// assign actuator mode
      AN    M    120.1;
      =     DB2740.DBX  105.4;
      =     DB2740.DBX  185.4;
      S     DB2740.DBX  265.4;
      =     DB2740.DBX  345.4;
      =     DB2740.DBX  425.4;
      =     DB2740.DBX  505.4;
      =     DB2740.DBX  585.4;
      =     DB2740.DBX  665.4;
      =     DB2740.DBX  745.4;
      =     DB2740.DBX  825.4;
      =     DB2740.DBX  905.4;
      =     DB2740.DBX  985.4;
      =     DB2740.DBX 1065.4;
      =     DB2740.DBX 1145.4;
      =     DB2740.DBX 1225.4;
      =     DB2740.DBX 1305.4;
      =     DB2740.DBX 1385.4;
      =     DB2740.DBX 1465.4;
      =     DB2740.DBX 1545.4;
      =     DB2740.DBX 1625.4;
      =     DB2740.DBX 1705.4;
      =     DB2740.DBX 1785.4;
      =     DB2740.DBX 1865.4;
      =     DB2740.DBX 1945.4;
      =     DB2740.DBX 2025.4;
      =     DB2740.DBX 2105.4;
      =     DB2740.DBX 2185.4;
      =     DB2740.DBX 2265.4;
      =     DB2740.DBX 2345.4;
      =     DB2740.DBX 2425.4;
      =     DB2740.DBX 2505.4;
      =     DB2740.DBX 2585.4;
      =     DB2740.DBX 2665.4;

MODE: SET   ;

NETWORK
TITLE =A14RRP1 Reinigungsrücklaufpumpe Anlage 14
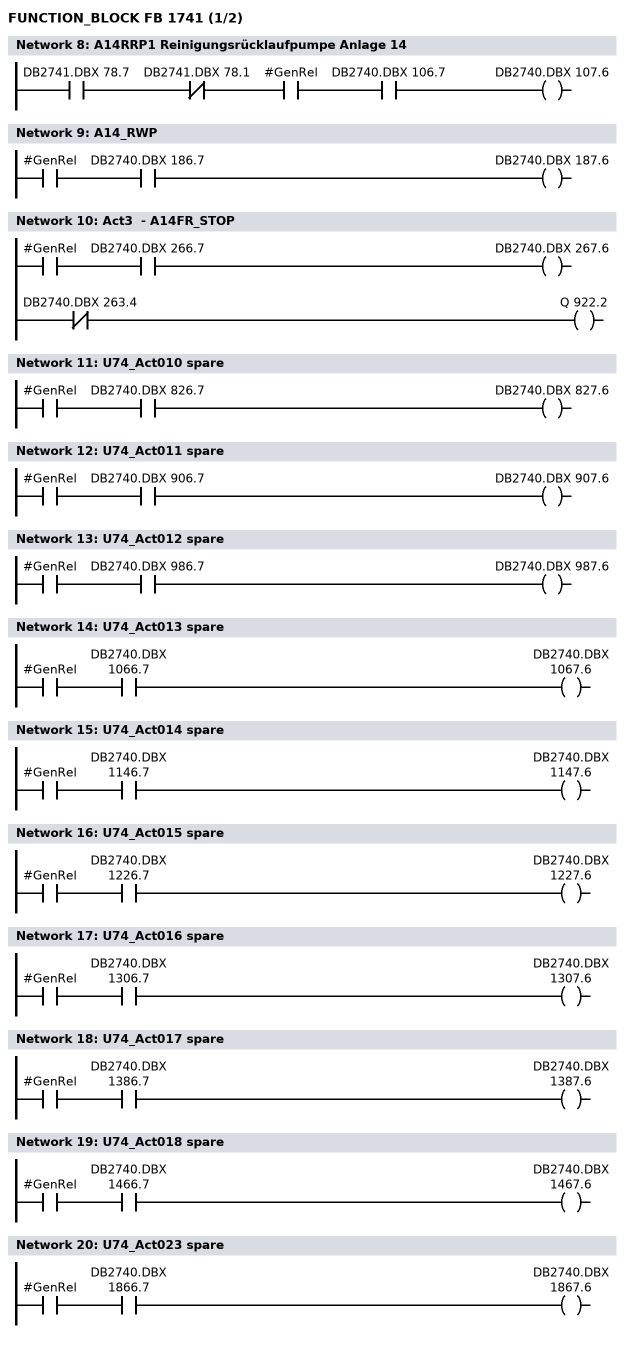

      A     DB2741.DBX   78.7;
      AN    DB2741.DBX   78.1;

      A     #GenRel;
      A     DB2740.DBX  106.7;
      =     DB2740.DBX  107.6;
NETWORK
TITLE =A14_RWP

      A     #GenRel;
      A     DB2740.DBX  186.7;
      =     DB2740.DBX  187.6;

NETWORK
TITLE =Act3  - A14FR_STOP

      A     #GenRel;
      A     DB2740.DBX  266.7;
      =     DB2740.DBX  267.6;

      AN    DB2740.DBX  263.4;
      =     Q    922.2;
NETWORK
TITLE =U74_Act010 spare

      A     #GenRel;
      A     DB2740.DBX  826.7;
      =     DB2740.DBX  827.6;
NETWORK
TITLE =U74_Act011 spare

      A     #GenRel;
      A     DB2740.DBX  906.7;
      =     DB2740.DBX  907.6;
NETWORK
TITLE =U74_Act012 spare

      A     #GenRel;
      A     DB2740.DBX  986.7;
      =     DB2740.DBX  987.6;
NETWORK
TITLE =U74_Act013 spare

      A     #GenRel;
      A     DB2740.DBX 1066.7;
      =     DB2740.DBX 1067.6;
NETWORK
TITLE =U74_Act014 spare

      A     #GenRel;
      A     DB2740.DBX 1146.7;
      =     DB2740.DBX 1147.6;
NETWORK
TITLE =U74_Act015 spare

      A     #GenRel;
      A     DB2740.DBX 1226.7;
      =     DB2740.DBX 1227.6;
NETWORK
TITLE =U74_Act016 spare

      A     #GenRel;
      A     DB2740.DBX 1306.7;
      =     DB2740.DBX 1307.6;
NETWORK
TITLE =U74_Act017 spare

      A     #GenRel;
      A     DB2740.DBX 1386.7;
      =     DB2740.DBX 1387.6;
NETWORK
TITLE =U74_Act018 spare

      A     #GenRel;
      A     DB2740.DBX 1466.7;
      =     DB2740.DBX 1467.6;
NETWORK
TITLE =U74_Act023 spare

      A     #GenRel;
      A     DB2740.DBX 1866.7;
      =     DB2740.DBX 1867.6;
NETWORK
TITLE =U74_Act024 spare
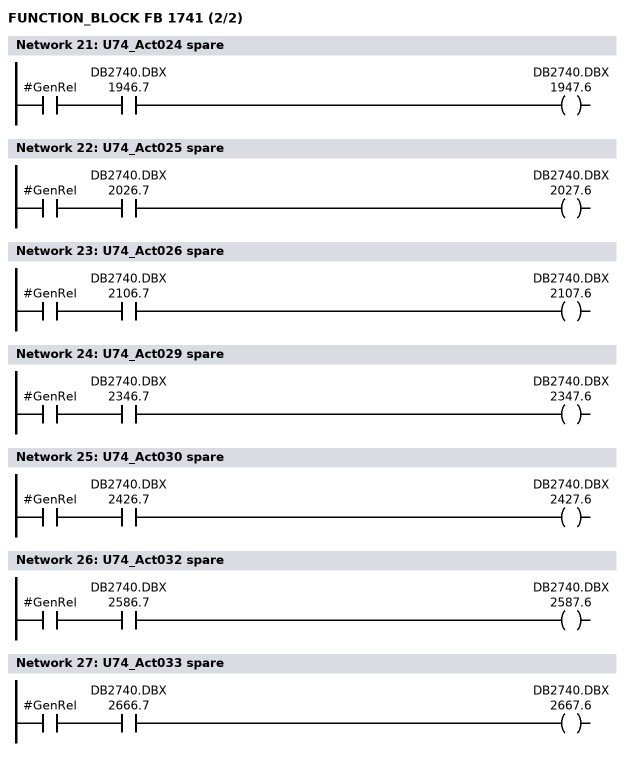

      A     #GenRel;
      A     DB2740.DBX 1946.7;
      =     DB2740.DBX 1947.6;
NETWORK
TITLE =U74_Act025 spare

      A     #GenRel;
      A     DB2740.DBX 2026.7;
      =     DB2740.DBX 2027.6;
NETWORK
TITLE =U74_Act026 spare

      A     #GenRel;
      A     DB2740.DBX 2106.7;
      =     DB2740.DBX 2107.6;
NETWORK
TITLE =U74_Act029 spare

      A     #GenRel;
      A     DB2740.DBX 2346.7;
      =     DB2740.DBX 2347.6;
NETWORK
TITLE =U74_Act030 spare

      A     #GenRel;
      A     DB2740.DBX 2426.7;
      =     DB2740.DBX 2427.6;
NETWORK
TITLE =U74_Act032 spare

      A     #GenRel;
      A     DB2740.DBX 2586.7;
      =     DB2740.DBX 2587.6;
NETWORK
TITLE =U74_Act033 spare

      A     #GenRel;
      A     DB2740.DBX 2666.7;
      =     DB2740.DBX 2667.6;
END_FUNCTION_BLOCK

FUNCTION_BLOCK FB 1770
TITLE =U077: KZE Anlage  3
FAMILY : BOTEC_F1
NAME : U077A
VERSION : 2.1


VAR_TEMP
  EStopOK : BOOL ;	//auxiliary flag
  CIP : BOOL ;	//CIP Program Selected
  xTmp : BOOL ;	//Temporary Bool(free for general use)
  DummyBool : BOOL ;	//Temporary Bool(free for general use)
  UnitNo : INT ;	//unit number
  UnitFB : INT ;	//unit expansion FB number
  rTmp : REAL ;	//Temporary REAL (free for general use)
  iTmp : INT ;	//Temporary INT (free for general use)
  DummyInt : INT ;	//Temporary INT (free for general use)
  dTmp : DINT ;	//Temporary DINT (free for general use)
END_VAR
BEGIN
NETWORK
TITLE =general

      CLR   ;
      =     #xTmp;
      =     #EStopOK;

      L     DB1770.DBW    0;
      T     #UnitNo;
      L     DB1770.DBW    2;
      T     #UnitFB;

NETWORK
TITLE =Universal value

      NOP   0;
// unv001 UnV 001 Process Status
      CALL FC    27 (
           UnitNo                   := #UnitNo,
           UnVRec                   := DB2775.unv001,
           ValExt                   := DB2775.DBD  234);

// unv002 UnV 002 Universal Value 02
      CALL FC    27 (
           UnitNo                   := #UnitNo,
           UnVRec                   := DB2775.unv002,
           ValExt                   := DB2775.DBD  362);

// unv003 UnV 003 Universal Value 03
      CALL FC    27 (
           UnitNo                   := #UnitNo,
           UnVRec                   := DB2775.unv003,
           ValExt                   := DB2775.DBD  490);

// unv004 UnV 004 Universal Value 04
      CALL FC    27 (
           UnitNo                   := #UnitNo,
           UnVRec                   := DB2775.unv004,
           ValExt                   := DB2775.DBD  618);

NETWORK
TITLE =special inputs

      NOP   0;
// KEG_MIXER_BOGEN_23_24 SpI 001 KEG Mixer/KZE Schwenkbogen
      CALL FC    14 (
           UnitNo                   := #UnitNo,
           SpIRec                   := DB2771.KEG_MIXER_BOGEN_23_24,
           SpIBit                   := I    950.0);

// KEG_MIXER_BOGEN_25_26 SpI 002 KEG Mixer/KZE Schwenkbogen
      CALL FC    14 (
           UnitNo                   := #UnitNo,
           SpIRec                   := DB2771.KEG_MIXER_BOGEN_25_26,
           SpIBit                   := I    950.1);

// KEG_MIXER_BOGEN_27_28 SpI 003 KEG Mixer/KZE Schwenkbogen
      CALL FC    14 (
           UnitNo                   := #UnitNo,
           SpIRec                   := DB2771.KEG_MIXER_BOGEN_27_28,
           SpIBit                   := I    950.2);

// KEG_MIXER_BOGEN_27_28_30 SpI 004 KEG Mixer/KZE Schwenkbogen
      CALL FC    14 (
           UnitNo                   := #UnitNo,
           SpIRec                   := DB2771.KEG_MIXER_BOGEN_27_28_30,
           SpIBit                   := I    950.3);

// KEG_MIXER_BOGEN_29_32 SpI 005 KEG Mixer/KZE Schwenkbogen
      CALL FC    14 (
           UnitNo                   := #UnitNo,
           SpIRec                   := DB2771.KEG_MIXER_BOGEN_29_32,
           SpIBit                   := I    950.4);

// KEG_MIXER_BOGEN_31_32 SpI 006 KEG Mixer/KZE Schwenkbogen
      CALL FC    14 (
           UnitNo                   := #UnitNo,
           SpIRec                   := DB2771.KEG_MIXER_BOGEN_31_32,
           SpIBit                   := I    950.5);

// KEG_MIXER_BOGEN_31_33 SpI 007 KEG Mixer/KZE Schwenkbogen
      CALL FC    14 (
           UnitNo                   := #UnitNo,
           SpIRec                   := DB2771.KEG_MIXER_BOGEN_31_33,
           SpIBit                   := I    950.6);

// KEG_MIXER_BOGEN_34_38 SpI 008 KEG Mixer/KZE Schwenkbogen
      CALL FC    14 (
           UnitNo                   := #UnitNo,
           SpIRec                   := DB2771.KEG_MIXER_BOGEN_34_38,
           SpIBit                   := I    950.7);

// KEG_MIXER_BOGEN_35_36_40 SpI 009 KEG Mixer/KZE Schwenkbogen
      CALL FC    14 (
           UnitNo                   := #UnitNo,
           SpIRec                   := DB2771.KEG_MIXER_BOGEN_35_36_40,
           SpIBit                   := I    951.0);

// KEG_MIXER_BOGEN_37_41 SpI 010 KEG Mixer/KZE Schwenkbogen
      CALL FC    14 (
           UnitNo                   := #UnitNo,
           SpIRec                   := DB2771.KEG_MIXER_BOGEN_37_41,
           SpIBit                   := I    951.1);

// KEG_MIXER_BOGEN_21_22 SpI 011 KEG Mixer/KZE Schwenkbogen
      CALL FC    14 (
           UnitNo                   := #UnitNo,
           SpIRec                   := DB2771.KEG_MIXER_BOGEN_21_22,
           SpIBit                   := I    951.2);

// KEG_MIXER_BOGEN_22_24 SpI 012 KEG Mixer/KZE Schwenkbogen
      CALL FC    14 (
           UnitNo                   := #UnitNo,
           SpIRec                   := DB2771.KEG_MIXER_BOGEN_22_24,
           SpIBit                   := I    951.3);

// KEG_MIXER_BOGEN_27_30 SpI 013 KEG Mixer/KZE Schwenkbogen
      CALL FC    14 (
           UnitNo                   := #UnitNo,
           SpIRec                   := DB2771.KEG_MIXER_BOGEN_27_30,
           SpIBit                   := I    951.4);

// KEG_MIXER_FRG_KZE SpI 014 KEG Mixer/KZE Freigabe CIP nur KZE
      CALL FC    14 (
           UnitNo                   := #UnitNo,
           SpIRec                   := DB2771.KEG_MIXER_FRG_KZE,
           SpIBit                   := I    947.0);

// KEG_MIXER_FRG_GES SpI 015 KEG Mixer/KZE Freigabe CIP Gesamt
      CALL FC    14 (
           UnitNo                   := #UnitNo,
           SpIRec                   := DB2771.KEG_MIXER_FRG_GES,
           SpIBit                   := I    946.6);

// KEG_MIXER_FRG_o_KZE SpI 016 KEG Mixer/KZE Freigabe CIP Gesamt ohne KZE
      CALL FC    14 (
           UnitNo                   := #UnitNo,
           SpIRec                   := DB2771.KEG_MIXER_FRG_o_KZE,
           SpIBit                   := I    946.7);

// KEG_MIXER_BOGEN_28_31 SpI 020 KEG Mixer/KZE Schwenkbogen
      CALL FC    14 (
           UnitNo                   := #UnitNo,
           SpIRec                   := DB2771.KEG_MIXER_BOGEN_28_31,
           SpIBit                   := I    951.5);

NETWORK
TITLE =messages

      NOP   0;
// msg001 Msg 001 Message 01
      CALL FC    16 (
           UnitNo                   := #UnitNo,
           MsgRec                   := DB2777.msg001,
           MsgBit                   := DB2777.DBX   82.7);

// msg002 Msg 002 Message 02
      CALL FC    16 (
           UnitNo                   := #UnitNo,
           MsgRec                   := DB2777.msg002,
           MsgBit                   := DB2777.DBX  142.7);

// msg003 Msg 003 Message 03
      CALL FC    16 (
           UnitNo                   := #UnitNo,
           MsgRec                   := DB2777.msg003,
           MsgBit                   := DB2777.DBX  202.7);

NETWORK
TITLE =unit supply

      UC    FB [#UnitFB];
END_FUNCTION_BLOCK

FUNCTION_BLOCK FB 1771
TITLE =U077: KZE Anlage  3
FAMILY : BOTEC_F1
NAME : U077E
VERSION : 1.2


VAR_TEMP
  CIP : BOOL ;	//CIP active
  UNIM : BOOL ;	//Unit Not In Maintenance
  GenRel : BOOL ;	//general OK (emergency and maintenance OK)
  EStopOK : BOOL ;	//emergency OK
  UnitNo : INT ;	//unit number
  xTmp : BOOL ;	//Temporary Bool
  iTmp : INT ;	//Temporary INT
  rTmp : REAL ;	//Temporary REAL
  dTmp : DINT ;	//Temporary DINT (free for general use)
  RetValInt : INT ;	//return value
END_VAR
BEGIN
NETWORK
TITLE =General

      SET   ;
// Simulation ---------------------------------------------------------------
      A     DB1771.DBX 1357.7;
      CC    FB  1779; // "U077Sim"
      A     DB1771.DBX   17.3;
      =     DB1771.DBX 1357.7; //Help bit for simulation

// get unit number ----------------------------------------------------------
      L     DB1770.DBW    0;
      T     #UnitNo;

// CIP ----------------------------------------------------------------------
      L     DB1771.DBD   54;
      L     0;
      <D    ;
      =     #CIP;

// emergency OK -------------------------------------------------------------
      A     DB1775.DBX   27.0; //Emergency Stop OK
      =     #EStopOK;

// Write Unit in Maintenance ------------------------------------------------

      AN    DB1771.DBX   69.7;
      =     #UNIM;

// emergency and maintenance OK ---------------------------------------------
      A     #EStopOK;
      A     #UNIM;
      =     #GenRel;

// communication ------------------------------------------------------------
      UC    FB  1775; // U077Com

NETWORK
TITLE =Universal Value

      NOP   0;

// ----------------------------------------------------------
// unv001 Process Status
// ----------------------------------------------------------
// process value to UnV
//      L     0.000000e+000
//      T     "U077UnVD".unv001.ValExt

// ----------------------------------------------------------
// unv002 Universal Value 02
// ----------------------------------------------------------
// process value to UnV
//      L     0.000000e+000
//      T     "U077UnVD".unv002.ValExt

// ----------------------------------------------------------
// unv003 Universal Value 03
// ----------------------------------------------------------
// process value to UnV
//      L     0.000000e+000
//      T     "U077UnVD".unv003.ValExt

// ----------------------------------------------------------
// unv004 Universal Value 04
// ----------------------------------------------------------
// process value to UnV
//      L     0.000000e+000
//      T     "U077UnVD".unv004.ValExt

NETWORK
TITLE =Special Input

      NOP   0;

// ----------------------------------------------------------
// KEG_MIXER_BOGEN_23_24 KEG Mixer/KZE Schwenkbogen
// ----------------------------------------------------------
//      SET
//      =     "U077SpID".KEG_MIXER_BOGEN_23_24.EAl
//      =     "U077SpID".KEG_MIXER_BOGEN_23_24.Pre

// ----------------------------------------------------------
// KEG_MIXER_BOGEN_25_26 KEG Mixer/KZE Schwenkbogen
// ----------------------------------------------------------
//      SET
//      =     "U077SpID".KEG_MIXER_BOGEN_25_26.EAl
//      =     "U077SpID".KEG_MIXER_BOGEN_25_26.Pre

// ----------------------------------------------------------
// KEG_MIXER_BOGEN_27_28 KEG Mixer/KZE Schwenkbogen
// ----------------------------------------------------------
//      SET
//      =     "U077SpID".KEG_MIXER_BOGEN_27_28.EAl
//      =     "U077SpID".KEG_MIXER_BOGEN_27_28.Pre

// ----------------------------------------------------------
// KEG_MIXER_BOGEN_27_28_30 KEG Mixer/KZE Schwenkbogen
// ----------------------------------------------------------
//      SET
//      =     "U077SpID".KEG_MIXER_BOGEN_27_28_30.EAl
//      =     "U077SpID".KEG_MIXER_BOGEN_27_28_30.Pre

// ----------------------------------------------------------
// KEG_MIXER_BOGEN_29_32 KEG Mixer/KZE Schwenkbogen
// ----------------------------------------------------------
//      SET
//      =     "U077SpID".KEG_MIXER_BOGEN_29_32.EAl
//      =     "U077SpID".KEG_MIXER_BOGEN_29_32.Pre

// ----------------------------------------------------------
// KEG_MIXER_BOGEN_31_32 KEG Mixer/KZE Schwenkbogen
// ----------------------------------------------------------
//      SET
//      =     "U077SpID".KEG_MIXER_BOGEN_31_32.EAl
//      =     "U077SpID".KEG_MIXER_BOGEN_31_32.Pre

// ----------------------------------------------------------
// KEG_MIXER_BOGEN_31_33 KEG Mixer/KZE Schwenkbogen
// ----------------------------------------------------------
//      SET
//      =     "U077SpID".KEG_MIXER_BOGEN_31_33.EAl
//      =     "U077SpID".KEG_MIXER_BOGEN_31_33.Pre

// ----------------------------------------------------------
// KEG_MIXER_BOGEN_34_38 KEG Mixer/KZE Schwenkbogen
// ----------------------------------------------------------
//      SET
//      =     "U077SpID".KEG_MIXER_BOGEN_34_38.EAl
//      =     "U077SpID".KEG_MIXER_BOGEN_34_38.Pre

// ----------------------------------------------------------
// KEG_MIXER_BOGEN_35_36_40 KEG Mixer/KZE Schwenkbogen
// ----------------------------------------------------------
//      SET
//      =     "U077SpID".KEG_MIXER_BOGEN_35_36_40.EAl
//      =     "U077SpID".KEG_MIXER_BOGEN_35_36_40.Pre

// ----------------------------------------------------------
// KEG_MIXER_BOGEN_37_41 KEG Mixer/KZE Schwenkbogen
// ----------------------------------------------------------
//      SET
//      =     "U077SpID".KEG_MIXER_BOGEN_37_41.EAl
//      =     "U077SpID".KEG_MIXER_BOGEN_37_41.Pre

// ----------------------------------------------------------
// KEG_MIXER_BOGEN_21_22 KEG Mixer/KZE Schwenkbogen
// ----------------------------------------------------------
//      SET
//      =     "U077SpID".KEG_MIXER_BOGEN_21_22.EAl
//      =     "U077SpID".KEG_MIXER_BOGEN_21_22.Pre

// ----------------------------------------------------------
// KEG_MIXER_BOGEN_22_24 KEG Mixer/KZE Schwenkbogen
// ----------------------------------------------------------
//      SET
//      =     "U077SpID".KEG_MIXER_BOGEN_22_24.EAl
//      =     "U077SpID".KEG_MIXER_BOGEN_22_24.Pre

// ----------------------------------------------------------
// KEG_MIXER_BOGEN_27_30 KEG Mixer/KZE Schwenkbogen
// ----------------------------------------------------------
//      SET
//      =     "U077SpID".KEG_MIXER_BOGEN_27_30.EAl
//      =     "U077SpID".KEG_MIXER_BOGEN_27_30.Pre

// ----------------------------------------------------------
// KEG_MIXER_FRG_KZE KEG Mixer/KZE Freigabe CIP nur KZE
// ----------------------------------------------------------
//      SET
//      =     "U077SpID".KEG_MIXER_FRG_KZE.EAl
//      =     "U077SpID".KEG_MIXER_FRG_KZE.Pre

// ----------------------------------------------------------
// KEG_MIXER_FRG_GES KEG Mixer/KZE Freigabe CIP Gesamt
// ----------------------------------------------------------
//      SET
//      =     "U077SpID".KEG_MIXER_FRG_GES.EAl
//      =     "U077SpID".KEG_MIXER_FRG_GES.Pre

// ----------------------------------------------------------
// KEG_MIXER_FRG_o_KZE KEG Mixer/KZE Freigabe CIP Gesamt ohne KZE
// ----------------------------------------------------------
//      SET
//      =     "U077SpID".KEG_MIXER_FRG_o_KZE.EAl
//      =     "U077SpID".KEG_MIXER_FRG_o_KZE.Pre

// ----------------------------------------------------------
// KEG_MIXER_BOGEN_28_31 KEG Mixer/KZE Schwenkbogen
// ----------------------------------------------------------
//      SET
//      =     "U077SpID".KEG_MIXER_BOGEN_28_31.EAl
//      =     "U077SpID".KEG_MIXER_BOGEN_28_31.Pre

NETWORK
TITLE =Messages

      NOP   0;

// ----------------------------------------------------------
// msg001 Message 01
// ----------------------------------------------------------
      SET   ;
      R     DB2777.DBX   80.7;
      =     DB2777.DBX   81.4;

      CLR   ;
      =     DB2777.DBX   82.7;

// ----------------------------------------------------------
// msg002 Message 02
// ----------------------------------------------------------
      SET   ;
      R     DB2777.DBX  140.7;
      =     DB2777.DBX  141.4;

      CLR   ;
      =     DB2777.DBX  142.7;

// ----------------------------------------------------------
// msg003 Message 03
// ----------------------------------------------------------
      SET   ;
      R     DB2777.DBX  200.7;
      =     DB2777.DBX  201.4;

      CLR   ;
      =     DB2777.DBX  202.7;

NETWORK
TITLE =Sequence organisation

      CLR   ;
      =     M    122.2;

// SFM supply ----------------------------------------------------------------

// sequencer ----------------------------------------------------------------
      A     DB1773.DBX   43.1;
      S     DB1773.DBX   97.3;

      CALL FC    40 (
           UnitNo                   := #UnitNo);

NETWORK
TITLE =Auto / Manual

      SET   ;
      AN    M    122.2;
      JC    MODE;
      AN    M    120.1;




MODE: SET   ;

END_FUNCTION_BLOCK

FUNCTION_BLOCK FB 1780
TITLE =U078: KZE Anlage  5
FAMILY : BOTEC_F1
NAME : U078A
VERSION : 2.1


VAR_TEMP
  EStopOK : BOOL ;	//auxiliary flag
  CIP : BOOL ;	//CIP Program Selected
  xTmp : BOOL ;	//Temporary Bool(free for general use)
  DummyBool : BOOL ;	//Temporary Bool(free for general use)
  UnitNo : INT ;	//unit number
  UnitFB : INT ;	//unit expansion FB number
  rTmp : REAL ;	//Temporary REAL (free for general use)
  iTmp : INT ;	//Temporary INT (free for general use)
  DummyInt : INT ;	//Temporary INT (free for general use)
  dTmp : DINT ;	//Temporary DINT (free for general use)
END_VAR
BEGIN
NETWORK
TITLE =general

      CLR   ;
      =     #xTmp;
      =     #EStopOK;

      L     DB1780.DBW    0;
      T     #UnitNo;
      L     DB1780.DBW    2;
      T     #UnitFB;

NETWORK
TITLE =analog inputs

      NOP   0;
// FIC450141 AnI 001
      CALL FC    24 (
           UnitNo                   := #UnitNo,
           AnIRec                   := DB2783.FIC450141,
           ValPer                   := #DummyInt);

// TIR450121 AnI 002
      CALL FC    24 (
           UnitNo                   := #UnitNo,
           AnIRec                   := DB2783.TIR450121,
           ValPer                   := #DummyInt);

// TIC450241 AnI 003
      CALL FC    24 (
           UnitNo                   := #UnitNo,
           AnIRec                   := DB2783.TIC450241,
           ValPer                   := #DummyInt);

// CIS450241 AnI 004
      CALL FC    24 (
           UnitNo                   := #UnitNo,
           AnIRec                   := DB2783.CIS450241,
           ValPer                   := #DummyInt);

// PIR450131 AnI 006
      CALL FC    24 (
           UnitNo                   := #UnitNo,
           AnIRec                   := DB2783.PIR450131,
           ValPer                   := #DummyInt);

NETWORK
TITLE =Universal value

      NOP   0;
// unv001 UnV 001 Process Status
      CALL FC    27 (
           UnitNo                   := #UnitNo,
           UnVRec                   := DB2785.unv001,
           ValExt                   := DB2785.DBD  234);

// unv002 UnV 002 Universal Value 02
      CALL FC    27 (
           UnitNo                   := #UnitNo,
           UnVRec                   := DB2785.unv002,
           ValExt                   := DB2785.DBD  362);

// unv003 UnV 003 Universal Value 03
      CALL FC    27 (
           UnitNo                   := #UnitNo,
           UnVRec                   := DB2785.unv003,
           ValExt                   := DB2785.DBD  490);

// unv004 UnV 004 Universal Value 04
      CALL FC    27 (
           UnitNo                   := #UnitNo,
           UnVRec                   := DB2785.unv004,
           ValExt                   := DB2785.DBD  618);

NETWORK
TITLE =special inputs

      NOP   0;
// KZE5_CIP_BEREIT SpI 003
      CALL FC    14 (
           UnitNo                   := #UnitNo,
           SpIRec                   := DB2781.KZE5_CIP_BEREIT,
           SpIBit                   := I    344.0);

// KZE5_PT_VOLL SpI 004
      CALL FC    14 (
           UnitNo                   := #UnitNo,
           SpIRec                   := DB2781.KZE5_PT_VOLL,
           SpIBit                   := I    344.2);

// KZE5_PT_LEER SpI 005
      CALL FC    14 (
           UnitNo                   := #UnitNo,
           SpIRec                   := DB2781.KZE5_PT_LEER,
           SpIBit                   := I    344.1);

// KZE5_BEREIT_F_KREISL SpI 006
      CALL FC    14 (
           UnitNo                   := #UnitNo,
           SpIRec                   := DB2781.KZE5_BEREIT_F_KREISL,
           SpIBit                   := I    344.5);

// KZE5_Watchdog SpI 007 KZE Anl.5 Watchdog
      CALL FC    14 (
           UnitNo                   := #UnitNo,
           SpIRec                   := DB2781.KZE5_Watchdog,
           SpIBit                   := I    345.7);

// KZE5_STERI_BEREIT SpI 009
      CALL FC    14 (
           UnitNo                   := #UnitNo,
           SpIRec                   := DB2781.KZE5_STERI_BEREIT,
           SpIBit                   := I    344.3);

// KZE5_AUSL_90GRAD SpI 010
      CALL FC    14 (
           UnitNo                   := #UnitNo,
           SpIRec                   := DB2781.KZE5_AUSL_90GRAD,
           SpIBit                   := I    344.4);

// KZE5_V720085 SpI 011 spare
      CALL FC    14 (
           UnitNo                   := #UnitNo,
           SpIRec                   := DB2781.KZE5_V720085,
           SpIBit                   := I    347.0);

// KZE5_LUFTWAESCHE_AKTIV SpI 012 Luftwäsche läuft
      CALL FC    14 (
           UnitNo                   := #UnitNo,
           SpIRec                   := DB2781.KZE5_LUFTWAESCHE_AKTIV,
           SpIBit                   := I    345.3);

// KZE5_LUFTWAESCHE_ENDE SpI 013 Luftwäsche beendet
      CALL FC    14 (
           UnitNo                   := #UnitNo,
           SpIRec                   := DB2781.KZE5_LUFTWAESCHE_ENDE,
           SpIBit                   := I    345.4);

// KZE5_FRG_KZE SpI 014 Freigabe CIP nur KZE
      CALL FC    14 (
           UnitNo                   := #UnitNo,
           SpIRec                   := DB2781.KZE5_FRG_KZE,
           SpIBit                   := I    344.6);

// KZE5_FRG_MIX_KZE_FUELL SpI 015 Freigabe CIP Mixer KZE Füller
      CALL FC    14 (
           UnitNo                   := #UnitNo,
           SpIRec                   := DB2781.KZE5_FRG_MIX_KZE_FUELL,
           SpIBit                   := I    344.7);

// KZE5_FRG_MIX_FUELL SpI 016 Freigabe CIP Mixer Füller
      CALL FC    14 (
           UnitNo                   := #UnitNo,
           SpIRec                   := DB2781.KZE5_FRG_MIX_FUELL,
           SpIBit                   := I    345.0);

// KZE5_V4500V03 SpI 017
      CALL FC    14 (
           UnitNo                   := #UnitNo,
           SpIRec                   := DB2781.KZE5_V4500V03,
           SpIBit                   := I    346.0);

// KZE5_V720015 SpI 018
      CALL FC    14 (
           UnitNo                   := #UnitNo,
           SpIRec                   := DB2781.KZE5_V720015,
           SpIBit                   := I    346.1);

// KZE5_V720016 SpI 019
      CALL FC    14 (
           UnitNo                   := #UnitNo,
           SpIRec                   := DB2781.KZE5_V720016,
           SpIBit                   := I    346.2);

// KZE5_V720017 SpI 020
      CALL FC    14 (
           UnitNo                   := #UnitNo,
           SpIRec                   := DB2781.KZE5_V720017,
           SpIBit                   := I    346.3);

// KZE5_V720081 SpI 021
      CALL FC    14 (
           UnitNo                   := #UnitNo,
           SpIRec                   := DB2781.KZE5_V720081,
           SpIBit                   := I    346.4);

// KZE5_V720082 SpI 022
      CALL FC    14 (
           UnitNo                   := #UnitNo,
           SpIRec                   := DB2781.KZE5_V720082,
           SpIBit                   := I    346.5);

// KZE5_V720083 SpI 023
      CALL FC    14 (
           UnitNo                   := #UnitNo,
           SpIRec                   := DB2781.KZE5_V720083,
           SpIBit                   := I    346.6);

// KZE5_V720084 SpI 024
      CALL FC    14 (
           UnitNo                   := #UnitNo,
           SpIRec                   := DB2781.KZE5_V720084,
           SpIBit                   := I    346.7);

// KZE5_V720086 SpI 025
      CALL FC    14 (
           UnitNo                   := #UnitNo,
           SpIRec                   := DB2781.KZE5_V720086,
           SpIBit                   := I    347.1);

// KZE5_V720087 SpI 026
      CALL FC    14 (
           UnitNo                   := #UnitNo,
           SpIRec                   := DB2781.KZE5_V720087,
           SpIBit                   := I    347.2);

// KZE5_V720182 SpI 027
      CALL FC    14 (
           UnitNo                   := #UnitNo,
           SpIRec                   := DB2781.KZE5_V720182,
           SpIBit                   := I    347.3);

// KZE5_V720006 SpI 028
      CALL FC    14 (
           UnitNo                   := #UnitNo,
           SpIRec                   := DB2781.KZE5_V720006,
           SpIBit                   := I    347.4);

NETWORK
TITLE =messages

      NOP   0;
// msg001 Msg 001 Message 01
      CALL FC    16 (
           UnitNo                   := #UnitNo,
           MsgRec                   := DB2787.msg001,
           MsgBit                   := DB2787.DBX   82.7);

// msg002 Msg 002 Message 02
      CALL FC    16 (
           UnitNo                   := #UnitNo,
           MsgRec                   := DB2787.msg002,
           MsgBit                   := DB2787.DBX  142.7);

// msg003 Msg 003 Message 03
      CALL FC    16 (
           UnitNo                   := #UnitNo,
           MsgRec                   := DB2787.msg003,
           MsgBit                   := DB2787.DBX  202.7);

NETWORK
TITLE =unit supply

      UC    FB [#UnitFB];
NETWORK
TITLE =KZE5_CIP_laeuft  KZE5 CIP Läuft
// Act 002
// Box           : KZE5
// Output address: Q344.0
      CALL FC    70 (
           UnitNo                   := #UnitNo,
           ActRec                   := DB2780.KZE5_CIP_laeuft,
           Typ                      := 0,
           FBa                      := #xTmp,
           FBa2                     := #xTmp,
           Out                      := Q    344.0);

NETWORK
TITLE =KZE5_CIP_ENDE  KZE5 CIP ENDE
// Act 003
// Box           : KZE5
// Output address: Q344.3
      CALL FC    70 (
           UnitNo                   := #UnitNo,
           ActRec                   := DB2780.KZE5_CIP_ENDE,
           Typ                      := 0,
           FBa                      := #xTmp,
           FBa2                     := #xTmp,
           Out                      := Q    344.3);

NETWORK
TITLE =KZE5_Medienwechsel  KZE5 Medienwechsel
// Act 004
// Box           : KZE5
// Output address: Q346.3
      CALL FC    70 (
           UnitNo                   := #UnitNo,
           ActRec                   := DB2780.KZE5_Medienwechsel,
           Typ                      := 0,
           FBa                      := #xTmp,
           FBa2                     := #xTmp,
           Out                      := Q    346.3);

NETWORK
TITLE =KZE5_Abpumpen  KZE5 Abpumpen
// Act 005
// Box           : KZE5
// Output address: Q344.6
      CALL FC    70 (
           UnitNo                   := #UnitNo,
           ActRec                   := DB2780.KZE5_Abpumpen,
           Typ                      := 0,
           FBa                      := #xTmp,
           FBa2                     := #xTmp,
           Out                      := Q    344.6);

NETWORK
TITLE =KZE5_KRSL_OA_PT  KZE5 Kreislauf ohne Ablauf Puffertank
// Act 006
// Box           : KZE5
// Output address: Q344.4
      CALL FC    70 (
           UnitNo                   := #UnitNo,
           ActRec                   := DB2780.KZE5_KRSL_OA_PT,
           Typ                      := 0,
           FBa                      := #xTmp,
           FBa2                     := #xTmp,
           Out                      := Q    344.4);

NETWORK
TITLE =KZE5_KRSL_MA_PT  KZE5 Kreislauf mit Ablauf Puffertank
// Act 007
// Box           : KZE5
// Output address: Q344.5
      CALL FC    70 (
           UnitNo                   := #UnitNo,
           ActRec                   := DB2780.KZE5_KRSL_MA_PT,
           Typ                      := 0,
           FBa                      := #xTmp,
           FBa2                     := #xTmp,
           Out                      := Q    344.5);

NETWORK
TITLE =KZE5_Grundstellung  KZE5 Grundstellung
// Act 008
// Box           : KZE5
// Output address: Q344.2
      CALL FC    70 (
           UnitNo                   := #UnitNo,
           ActRec                   := DB2780.KZE5_Grundstellung,
           Typ                      := 0,
           FBa                      := #xTmp,
           FBa2                     := #xTmp,
           Out                      := Q    344.2);

NETWORK
TITLE =KZE5_Heizung_ein  KZE5 Heizung ein
// Act 012
// Box           : KZE5
// Output address: Q344.1
      CALL FC    70 (
           UnitNo                   := #UnitNo,
           ActRec                   := DB2780.KZE5_Heizung_ein,
           Typ                      := 0,
           FBa                      := #xTmp,
           FBa2                     := #xTmp,
           Out                      := Q    344.1);

NETWORK
TITLE =KZE5_H2O  KZE5 Hauptschritte Wasser
// Act 013
// Box           : KZE5
// Output address: Q345.1
      CALL FC    70 (
           UnitNo                   := #UnitNo,
           ActRec                   := DB2780.KZE5_H2O,
           Typ                      := 0,
           FBa                      := #xTmp,
           FBa2                     := #xTmp,
           Out                      := Q    345.1);

NETWORK
TITLE =KZE5_Lauge  KZE5 Lauge Kreislauf
// Act 014
// Box           : KZE5
// Output address: Q345.2
      CALL FC    70 (
           UnitNo                   := #UnitNo,
           ActRec                   := DB2780.KZE5_Lauge,
           Typ                      := 0,
           FBa                      := #xTmp,
           FBa2                     := #xTmp,
           Out                      := Q    345.2);

NETWORK
TITLE =KZE5_Saeure  KZE5 Säure Kreislauf
// Act 015
// Box           : KZE5
// Output address: Q345.3
      CALL FC    70 (
           UnitNo                   := #UnitNo,
           ActRec                   := DB2780.KZE5_Saeure,
           Typ                      := 0,
           FBa                      := #xTmp,
           FBa2                     := #xTmp,
           Out                      := Q    345.3);

NETWORK
TITLE =KZE5_Sterilisation  KZE5 Sterilisation angewählt
// Act 016
// Box           : KZE5
// Output address: Q345.4
      CALL FC    70 (
           UnitNo                   := #UnitNo,
           ActRec                   := DB2780.KZE5_Sterilisation,
           Typ                      := 0,
           FBa                      := #xTmp,
           FBa2                     := #xTmp,
           Out                      := Q    345.4);

NETWORK
TITLE =KZE5_Abkuehlen  KZE5 Abkühlen
// Act 017
// Box           : KZE5
// Output address: Q345.5
      CALL FC    70 (
           UnitNo                   := #UnitNo,
           ActRec                   := DB2780.KZE5_Abkuehlen,
           Typ                      := 0,
           FBa                      := #xTmp,
           FBa2                     := #xTmp,
           Out                      := Q    345.5);

NETWORK
TITLE =KZE5_Freiabe_Luftwaesche  KZE5 Freigabe Luftwäsche
// Act 020
// Box           : KZE5
// Output address: Q346.4
      CALL FC    70 (
           UnitNo                   := #UnitNo,
           ActRec                   := DB2780.KZE5_Freiabe_Luftwaesche,
           Typ                      := 0,
           FBa                      := #xTmp,
           FBa2                     := #xTmp,
           Out                      := Q    346.4);

END_FUNCTION_BLOCK

FUNCTION_BLOCK FB 1781
TITLE =U078: KZE Anlage  5
FAMILY : BOTEC_F1
NAME : U078E
VERSION : 1.2


VAR_TEMP
  CIP : BOOL ;	//CIP active
  UNIM : BOOL ;	//Unit Not In Maintenance
  GenRel : BOOL ;	//general OK (emergency and maintenance OK)
  EStopOK : BOOL ;	//emergency OK
  UnitNo : INT ;	//unit number
  xTmp : BOOL ;	//Temporary Bool
  iTmp : INT ;	//Temporary INT
  rTmp : REAL ;	//Temporary REAL
  dTmp : DINT ;	//Temporary DINT (free for general use)
  RetValInt : INT ;	//return value
END_VAR
BEGIN
NETWORK
TITLE =General

      SET   ;
// Simulation ---------------------------------------------------------------
      A     DB1781.DBX 1357.7;
      CC    FB  1789; // "U078Sim"
      A     DB1781.DBX   17.3;
      =     DB1781.DBX 1357.7; //Help bit for simulation

// get unit number ----------------------------------------------------------
      L     DB1780.DBW    0;
      T     #UnitNo;

// CIP ----------------------------------------------------------------------
      L     DB1781.DBD   54;
      L     0;
      <D    ;
      =     #CIP;

// emergency OK -------------------------------------------------------------
      A     DB1785.DBX   27.0; //Emergency Stop OK
      =     #EStopOK;

// Write Unit in Maintenance ------------------------------------------------

      AN    DB1781.DBX   69.7;
      =     #UNIM;

// emergency and maintenance OK ---------------------------------------------
      A     #EStopOK;
      A     #UNIM;
      =     #GenRel;

// communication ------------------------------------------------------------
      UC    FB  1785; // U078Com

NETWORK
TITLE =Analog Inputs

      NOP   0;

// ----------------------------------------------------------
// FIC450141
// ----------------------------------------------------------


      L     ID   348; // FIC
      L     1.000000e+001;
      /R    ;

      T     DB2783.DBD  214;
      SET   ;
      =     DB2783.DBX  143.5;

      L     DB1781.DBD 1118; // !!! insert correct SFM !!!
      T     DB2783.DBD  238;

      SET   ;
      =     DB2783.DBX  141.5;

// ----------------------------------------------------------
// TIR450121
// ----------------------------------------------------------
      L     ID   352; //TIR
      T     DB2783.DBD  334;
      SET   ;
      =     DB2783.DBX  263.5;

      L     DB1781.DBD 1118; // !!! insert correct SFM !!!
      T     DB2783.DBD  358;

      SET   ;
      =     DB2783.DBX  261.5;

// ----------------------------------------------------------
// TIC450241
// ----------------------------------------------------------
      L     ID   360; //TIC
      T     DB2783.DBD  454;
      SET   ;
      =     DB2783.DBX  383.5;

      L     DB1781.DBD 1118; // !!! insert correct SFM !!!
      T     DB2783.DBD  478;

      SET   ;
      =     DB2783.DBX  381.5;

// ----------------------------------------------------------
// CIS450241
// ----------------------------------------------------------
      L     ID   364; // CIS
      T     DB2783.DBD  574;
      SET   ;
      =     DB2783.DBX  503.5;

      L     DB1781.DBD 1118; // !!! insert correct SFM !!!
      T     DB2783.DBD  598;

      SET   ;
      =     DB2783.DBX  501.5;

// ----------------------------------------------------------
// PIR450131
// ----------------------------------------------------------
      L     ID   356; // PIR
      T     DB2783.DBD  814;
      SET   ;
      =     DB2783.DBX  743.5;

      L     DB1781.DBD 1118; // !!! insert correct SFM !!!
      T     DB2783.DBD  838;

      SET   ;
      =     DB2783.DBX  741.5;

NETWORK
TITLE =Universal Value

      NOP   0;

// ----------------------------------------------------------
// unv001 Process Status
// ----------------------------------------------------------
// process value to UnV
//      L     0.000000e+000
//      T     "U078UnVD".unv001.ValExt

// ----------------------------------------------------------
// unv002 Universal Value 02
// ----------------------------------------------------------
// process value to UnV
//      L     0.000000e+000
//      T     "U078UnVD".unv002.ValExt

// ----------------------------------------------------------
// unv003 Universal Value 03
// ----------------------------------------------------------
// process value to UnV
//      L     0.000000e+000
//      T     "U078UnVD".unv003.ValExt

// ----------------------------------------------------------
// unv004 Universal Value 04
// ----------------------------------------------------------
// process value to UnV
//      L     0.000000e+000
//      T     "U078UnVD".unv004.ValExt

NETWORK
TITLE =Special Input

      NOP   0;

// ----------------------------------------------------------
// KZE5_CIP_BEREIT
// ----------------------------------------------------------
//      CLR
//      =     "U078SpID".KZE5_CIP_BEREIT.EAl
//      =     "U078SpID".KZE5_CIP_BEREIT.Pre

// ----------------------------------------------------------
// KZE5_PT_VOLL
// ----------------------------------------------------------
//      CLR
//      =     "U078SpID".KZE5_PT_VOLL.EAl
//      =     "U078SpID".KZE5_PT_VOLL.Pre

// ----------------------------------------------------------
// KZE5_PT_LEER
// ----------------------------------------------------------
//      CLR
//      =     "U078SpID".KZE5_PT_LEER.EAl
//      =     "U078SpID".KZE5_PT_LEER.Pre

// ----------------------------------------------------------
// KZE5_BEREIT_F_KREISL
// ----------------------------------------------------------
//      CLR
//      =     "U078SpID".KZE5_BEREIT_F_KREISL.EAl
//      =     "U078SpID".KZE5_BEREIT_F_KREISL.Pre

// ----------------------------------------------------------
// KZE5_Watchdog KZE Anl.5 Watchdog
// ----------------------------------------------------------
//      CLR
//      =     "U078SpID".KZE5_Watchdog.EAl
//      =     "U078SpID".KZE5_Watchdog.Pre

// ----------------------------------------------------------
// KZE5_STERI_BEREIT
// ----------------------------------------------------------
//      CLR
//      =     "U078SpID".KZE5_STERI_BEREIT.EAl
//      =     "U078SpID".KZE5_STERI_BEREIT.Pre

// ----------------------------------------------------------
// KZE5_AUSL_90GRAD
// ----------------------------------------------------------
//      CLR
//      =     "U078SpID".KZE5_AUSL_90GRAD.EAl
//      =     "U078SpID".KZE5_AUSL_90GRAD.Pre

// ----------------------------------------------------------
// KZE5_V720085 spare
// ----------------------------------------------------------
//      CLR
//      =     "U078SpID".KZE5_V720085.EAl
//      =     "U078SpID".KZE5_V720085.Pre

// ----------------------------------------------------------
// KZE5_LUFTWAESCHE_AKTIV Luftwäsche läuft
// ----------------------------------------------------------
//      CLR
//      =     "U078SpID".KZE5_LUFTWAESCHE_AKTIV.EAl
//      =     "U078SpID".KZE5_LUFTWAESCHE_AKTIV.Pre

// ----------------------------------------------------------
// KZE5_LUFTWAESCHE_ENDE Luftwäsche beendet
// ----------------------------------------------------------
//      CLR
//      =     "U078SpID".KZE5_LUFTWAESCHE_ENDE.EAl
//      =     "U078SpID".KZE5_LUFTWAESCHE_ENDE.Pre

// ----------------------------------------------------------
// KZE5_FRG_KZE Freigabe CIP nur KZE
// ----------------------------------------------------------
//      CLR
//      =     "U078SpID".KZE5_FRG_KZE.EAl
//      =     "U078SpID".KZE5_FRG_KZE.Pre

// ----------------------------------------------------------
// KZE5_FRG_MIX_KZE_FUELL Freigabe CIP Mixer KZE Füller
// ----------------------------------------------------------
//      CLR
//      =     "U078SpID".KZE5_FRG_MIX_KZE_FUELL.EAl
//      =     "U078SpID".KZE5_FRG_MIX_KZE_FUELL.Pre

// ----------------------------------------------------------
// KZE5_FRG_MIX_FUELL Freigabe CIP Mixer Füller
// ----------------------------------------------------------
//      CLR
//      =     "U078SpID".KZE5_FRG_MIX_FUELL.EAl
//      =     "U078SpID".KZE5_FRG_MIX_FUELL.Pre

// ----------------------------------------------------------
// KZE5_V4500V03
// ----------------------------------------------------------
//      CLR
//      =     "U078SpID".KZE5_V4500V03.EAl
//      =     "U078SpID".KZE5_V4500V03.Pre

// ----------------------------------------------------------
// KZE5_V720015
// ----------------------------------------------------------
//      CLR
//      =     "U078SpID".KZE5_V720015.EAl
//      =     "U078SpID".KZE5_V720015.Pre

// ----------------------------------------------------------
// KZE5_V720016
// ----------------------------------------------------------
//      CLR
//      =     "U078SpID".KZE5_V720016.EAl
//      =     "U078SpID".KZE5_V720016.Pre

// ----------------------------------------------------------
// KZE5_V720017
// ----------------------------------------------------------
//      CLR
//      =     "U078SpID".KZE5_V720017.EAl
//      =     "U078SpID".KZE5_V720017.Pre

// ----------------------------------------------------------
// KZE5_V720081
// ----------------------------------------------------------
//      CLR
//      =     "U078SpID".KZE5_V720081.EAl
//      =     "U078SpID".KZE5_V720081.Pre

// ----------------------------------------------------------
// KZE5_V720082
// ----------------------------------------------------------
//      CLR
//      =     "U078SpID".KZE5_V720082.EAl
//      =     "U078SpID".KZE5_V720082.Pre

// ----------------------------------------------------------
// KZE5_V720083
// ----------------------------------------------------------
//      CLR
//      =     "U078SpID".KZE5_V720083.EAl
//      =     "U078SpID".KZE5_V720083.Pre

// ----------------------------------------------------------
// KZE5_V720084
// ----------------------------------------------------------
//      CLR
//      =     "U078SpID".KZE5_V720084.EAl
//      =     "U078SpID".KZE5_V720084.Pre

// ----------------------------------------------------------
// KZE5_V720086
// ----------------------------------------------------------
//      CLR
//      =     "U078SpID".KZE5_V720086.EAl
//      =     "U078SpID".KZE5_V720086.Pre

// ----------------------------------------------------------
// KZE5_V720087
// ----------------------------------------------------------
//      CLR
//      =     "U078SpID".KZE5_V720087.EAl
//      =     "U078SpID".KZE5_V720087.Pre

// ----------------------------------------------------------
// KZE5_V720182
// ----------------------------------------------------------
//      CLR
//      =     "U078SpID".KZE5_V720182.EAl
//      =     "U078SpID".KZE5_V720182.Pre

// ----------------------------------------------------------
// KZE5_V720006
// ----------------------------------------------------------
//      CLR
//      =     "U078SpID".KZE5_V720006.EAl
//      =     "U078SpID".KZE5_V720006.Pre

NETWORK
TITLE =Messages

      NOP   0;

// ----------------------------------------------------------
// msg001 Message 01
// ----------------------------------------------------------
      SET   ;
      R     DB2787.DBX   80.7;
      =     DB2787.DBX   81.4;

      CLR   ;
      =     DB2787.DBX   82.7;

// ----------------------------------------------------------
// msg002 Message 02
// ----------------------------------------------------------
      SET   ;
      R     DB2787.DBX  140.7;
      =     DB2787.DBX  141.4;

      CLR   ;
      =     DB2787.DBX  142.7;

// ----------------------------------------------------------
// msg003 Message 03
// ----------------------------------------------------------
      SET   ;
      R     DB2787.DBX  200.7;
      =     DB2787.DBX  201.4;

      CLR   ;
      =     DB2787.DBX  202.7;

NETWORK
TITLE =Sequence organisation

      CLR   ;
      =     M    122.2;

// SFM supply ----------------------------------------------------------------

// analog value to SFM  -----------------------
      L     DB2783.DBD  146;
      T     DB1781.DBD 1122;

// analog value to SFM  -----------------------
      L     DB2783.DBD  266;
      T     DB1781.DBD 1122;

// analog value to SFM  -----------------------
      L     DB2783.DBD  386;
      T     DB1781.DBD 1122;

// analog value to SFM  -----------------------
      L     DB2783.DBD  506;
      T     DB1781.DBD 1122;

// analog value to SFM  -----------------------
      L     DB2783.DBD  746;
      T     DB1781.DBD 1122;

// CIP Counter
      CALL FC    29 (
           UnitNo                   := #UnitNo,
           Value                    := DB1785.DBD  138,
           Enable                   := TRUE,
           Down                     := FALSE,
           OriginDetect             := 0.000000e+000,
           MaxDiffPS                := 1.000000e+000,
           SFMRec                   := DB1781.Seq.SFM[15],
           ValueOld                 := DB1781.DBD 1418);

// sequencer ----------------------------------------------------------------
      A     DB1783.DBX   43.1;
      S     DB1783.DBX   97.3;

      CALL FC    40 (
           UnitNo                   := #UnitNo);

NETWORK
TITLE =Auto / Manual

      SET   ;
      AN    M    122.2;
      JC    MODE;
      AN    M    120.1;

// assign actuator mode
      AN    M    120.1;
      =     DB2780.DBX  185.4;
      =     DB2780.DBX  265.4;
      =     DB2780.DBX  345.4;
      =     DB2780.DBX  425.4;
      =     DB2780.DBX  505.4;
      =     DB2780.DBX  585.4;
      =     DB2780.DBX  665.4;
      =     DB2780.DBX  985.4;
      =     DB2780.DBX 1065.4;
      =     DB2780.DBX 1145.4;
      =     DB2780.DBX 1225.4;
      =     DB2780.DBX 1305.4;
      =     DB2780.DBX 1385.4;
      =     DB2780.DBX 1625.4;



MODE: SET   ;

NETWORK
TITLE =KZE5_CIP_laeuft KZE5 CIP Läuft
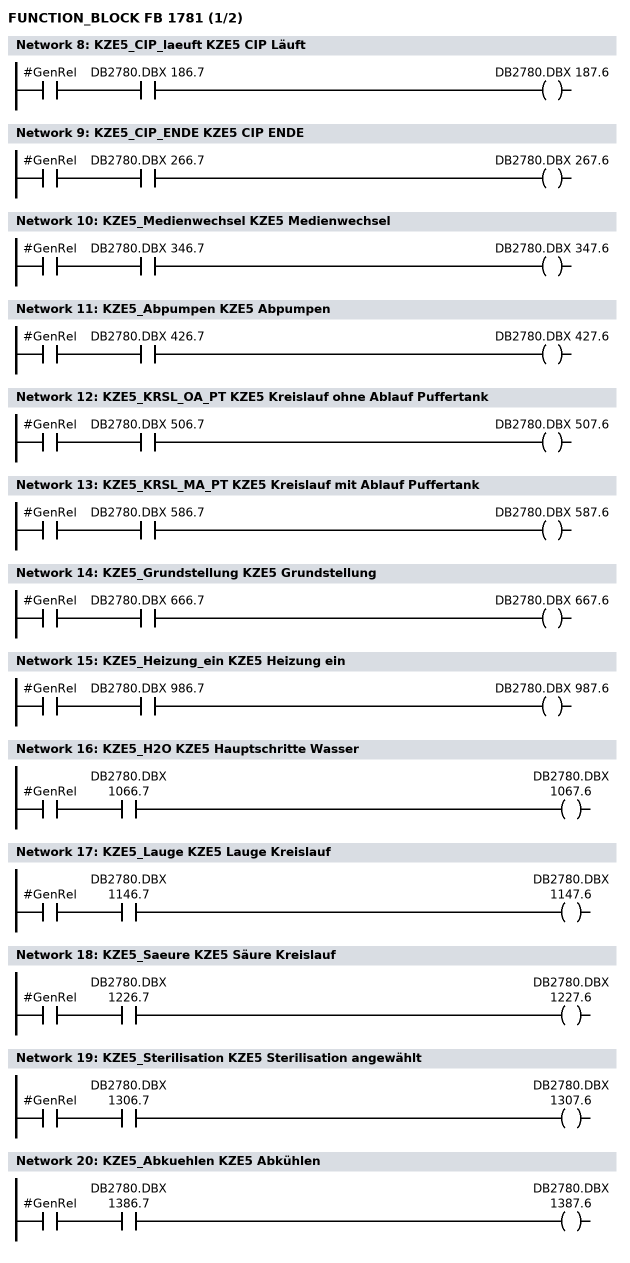

      A     #GenRel;
      A     DB2780.DBX  186.7;
      =     DB2780.DBX  187.6;
NETWORK
TITLE =KZE5_CIP_ENDE KZE5 CIP ENDE

      A     #GenRel;
      A     DB2780.DBX  266.7;
      =     DB2780.DBX  267.6;
NETWORK
TITLE =KZE5_Medienwechsel KZE5 Medienwechsel

      A     #GenRel;
      A     DB2780.DBX  346.7;
      =     DB2780.DBX  347.6;
NETWORK
TITLE =KZE5_Abpumpen KZE5 Abpumpen

      A     #GenRel;
      A     DB2780.DBX  426.7;
      =     DB2780.DBX  427.6;
NETWORK
TITLE =KZE5_KRSL_OA_PT KZE5 Kreislauf ohne Ablauf Puffertank

      A     #GenRel;
      A     DB2780.DBX  506.7;
      =     DB2780.DBX  507.6;
NETWORK
TITLE =KZE5_KRSL_MA_PT KZE5 Kreislauf mit Ablauf Puffertank

      A     #GenRel;
      A     DB2780.DBX  586.7;
      =     DB2780.DBX  587.6;
NETWORK
TITLE =KZE5_Grundstellung KZE5 Grundstellung

      A     #GenRel;
      A     DB2780.DBX  666.7;
      =     DB2780.DBX  667.6;
NETWORK
TITLE =KZE5_Heizung_ein KZE5 Heizung ein

      A     #GenRel;
      A     DB2780.DBX  986.7;
      =     DB2780.DBX  987.6;
NETWORK
TITLE =KZE5_H2O KZE5 Hauptschritte Wasser

      A     #GenRel;
      A     DB2780.DBX 1066.7;
      =     DB2780.DBX 1067.6;
NETWORK
TITLE =KZE5_Lauge KZE5 Lauge Kreislauf

      A     #GenRel;
      A     DB2780.DBX 1146.7;
      =     DB2780.DBX 1147.6;
NETWORK
TITLE =KZE5_Saeure KZE5 Säure Kreislauf

      A     #GenRel;
      A     DB2780.DBX 1226.7;
      =     DB2780.DBX 1227.6;
NETWORK
TITLE =KZE5_Sterilisation KZE5 Sterilisation angewählt

      A     #GenRel;
      A     DB2780.DBX 1306.7;
      =     DB2780.DBX 1307.6;
NETWORK
TITLE =KZE5_Abkuehlen KZE5 Abkühlen

      A     #GenRel;
      A     DB2780.DBX 1386.7;
      =     DB2780.DBX 1387.6;
NETWORK
TITLE =KZE5_Freiabe_Luftwaesche KZE5 Freigabe Luftwäsche
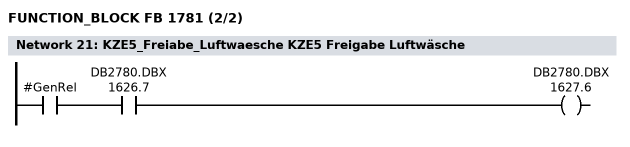

      A     #GenRel;
      A     DB2780.DBX 1626.7;
      =     DB2780.DBX 1627.6;
END_FUNCTION_BLOCK

FUNCTION_BLOCK FB 1790
TITLE =U079: KZE Anlage 14
FAMILY : BOTEC_F1
NAME : U079A
VERSION : 2.1


VAR_TEMP
  EStopOK : BOOL ;	//auxiliary flag
  CIP : BOOL ;	//CIP Program Selected
  xTmp : BOOL ;	//Temporary Bool(free for general use)
  DummyBool : BOOL ;	//Temporary Bool(free for general use)
  UnitNo : INT ;	//unit number
  UnitFB : INT ;	//unit expansion FB number
  rTmp : REAL ;	//Temporary REAL (free for general use)
  iTmp : INT ;	//Temporary INT (free for general use)
  DummyInt : INT ;	//Temporary INT (free for general use)
  dTmp : DINT ;	//Temporary DINT (free for general use)
END_VAR
BEGIN
NETWORK
TITLE =general

      CLR   ;
      =     #xTmp;
      =     #EStopOK;

      L     DB1790.DBW    0;
      T     #UnitNo;
      L     DB1790.DBW    2;
      T     #UnitFB;

NETWORK
TITLE =analog inputs

      NOP   0;
// A14_KZE_FIC7101 AnI 001
      CALL FC    24 (
           UnitNo                   := #UnitNo,
           AnIRec                   := DB2793.A14_KZE_FIC7101,
           ValPer                   := PIW 1006);

// A14_KZE_TIR7101 AnI 002
      CALL FC    24 (
           UnitNo                   := #UnitNo,
           AnIRec                   := DB2793.A14_KZE_TIR7101,
           ValPer                   := PIW 1010);

// A14_KZE_TIC7102 AnI 003
      CALL FC    24 (
           UnitNo                   := #UnitNo,
           AnIRec                   := DB2793.A14_KZE_TIC7102,
           ValPer                   := PIW 1014);

// A14_KZE_CIS7102 AnI 004
      CALL FC    24 (
           UnitNo                   := #UnitNo,
           AnIRec                   := DB2793.A14_KZE_CIS7102,
           ValPer                   := PIW 1018);

// A14_KZE_TIS7111 AnI 005
      CALL FC    24 (
           UnitNo                   := #UnitNo,
           AnIRec                   := DB2793.A14_KZE_TIS7111,
           ValPer                   := PIW 1022);

NETWORK
TITLE =Universal value

      NOP   0;
// unv001 UnV 001 Process Status
      CALL FC    27 (
           UnitNo                   := #UnitNo,
           UnVRec                   := DB2795.unv001,
           ValExt                   := DB2795.DBD  234);

// unv002 UnV 002 Universal Value 02
      CALL FC    27 (
           UnitNo                   := #UnitNo,
           UnVRec                   := DB2795.unv002,
           ValExt                   := DB2795.DBD  362);

// unv003 UnV 003 Universal Value 03
      CALL FC    27 (
           UnitNo                   := #UnitNo,
           UnVRec                   := DB2795.unv003,
           ValExt                   := DB2795.DBD  490);

// unv004 UnV 004 Universal Value 04
      CALL FC    27 (
           UnitNo                   := #UnitNo,
           UnVRec                   := DB2795.unv004,
           ValExt                   := DB2795.DBD  618);

NETWORK
TITLE =special inputs

      NOP   0;
// KZE14_CIP_BEREIT SpI 003
      CALL FC    14 (
           UnitNo                   := #UnitNo,
           SpIRec                   := DB2791.KZE14_CIP_BEREIT,
           SpIBit                   := I   1002.0);

// KZE14_PT_VOLL SpI 004
      CALL FC    14 (
           UnitNo                   := #UnitNo,
           SpIRec                   := DB2791.KZE14_PT_VOLL,
           SpIBit                   := I   1002.2);

// KZE14_PT_LEER SpI 005
      CALL FC    14 (
           UnitNo                   := #UnitNo,
           SpIRec                   := DB2791.KZE14_PT_LEER,
           SpIBit                   := I   1002.1);

// KZE14_BEREIT_F_KREISL SpI 006
      CALL FC    14 (
           UnitNo                   := #UnitNo,
           SpIRec                   := DB2791.KZE14_BEREIT_F_KREISL,
           SpIBit                   := I   1002.5);

// KZE14_STERI_BEREIT SpI 009
      CALL FC    14 (
           UnitNo                   := #UnitNo,
           SpIRec                   := DB2791.KZE14_STERI_BEREIT,
           SpIBit                   := I   1002.3);

// KZE14_AUSL_90GRAD SpI 010
      CALL FC    14 (
           UnitNo                   := #UnitNo,
           SpIRec                   := DB2791.KZE14_AUSL_90GRAD,
           SpIBit                   := I   1002.4);

// KZE14_FRG_KZE SpI 014 Freigabe CIP nur KZE
      CALL FC    14 (
           UnitNo                   := #UnitNo,
           SpIRec                   := DB2791.KZE14_FRG_KZE,
           SpIBit                   := I   1002.6);

// KZE14_FRG_MIX_KZE_FUEL SpI 015 Freigabe CIP Mixer KZE Füller
      CALL FC    14 (
           UnitNo                   := #UnitNo,
           SpIRec                   := DB2791.KZE14_FRG_MIX_KZE_FUEL,
           SpIBit                   := I   1002.7);

// KZE14_FRG_MIX_FUEL SpI 016 Freigabe CIP Mixer Füller
      CALL FC    14 (
           UnitNo                   := #UnitNo,
           SpIRec                   := DB2791.KZE14_FRG_MIX_FUEL,
           SpIBit                   := I   1003.0);

// KZE14_FRG_KZE_FUEL SpI 017 Freigabe CIP KZE Füller
      CALL FC    14 (
           UnitNo                   := #UnitNo,
           SpIRec                   := DB2791.KZE14_FRG_KZE_FUEL,
           SpIBit                   := I   1003.1);

// KZE14_V710021 SpI 020 Ventil
      CALL FC    14 (
           UnitNo                   := #UnitNo,
           SpIRec                   := DB2791.KZE14_V710021,
           SpIBit                   := I   1004.0);

// KZE14_V710131 SpI 021 Ventil
      CALL FC    14 (
           UnitNo                   := #UnitNo,
           SpIRec                   := DB2791.KZE14_V710131,
           SpIBit                   := I   1004.1);

// KZE14_V710005 SpI 022 Ventil
      CALL FC    14 (
           UnitNo                   := #UnitNo,
           SpIRec                   := DB2791.KZE14_V710005,
           SpIBit                   := I   1004.2);

// KZE14_V710181 SpI 023 Ventil
      CALL FC    14 (
           UnitNo                   := #UnitNo,
           SpIRec                   := DB2791.KZE14_V710181,
           SpIBit                   := I   1004.3);

// KZE14_V710182 SpI 024 Ventil
      CALL FC    14 (
           UnitNo                   := #UnitNo,
           SpIRec                   := DB2791.KZE14_V710182,
           SpIBit                   := I   1004.4);

// KZE14_V813101 SpI 025 Ventil
      CALL FC    14 (
           UnitNo                   := #UnitNo,
           SpIRec                   := DB2791.KZE14_V813101,
           SpIBit                   := I   1004.5);

// KZE14_V813102 SpI 026 Ventil
      CALL FC    14 (
           UnitNo                   := #UnitNo,
           SpIRec                   := DB2791.KZE14_V813102,
           SpIBit                   := I   1004.6);

// KZE14_V812101 SpI 027 Ventil
      CALL FC    14 (
           UnitNo                   := #UnitNo,
           SpIRec                   := DB2791.KZE14_V812101,
           SpIBit                   := I   1004.7);

// KZE14_V812102 SpI 028 Ventil
      CALL FC    14 (
           UnitNo                   := #UnitNo,
           SpIRec                   := DB2791.KZE14_V812102,
           SpIBit                   := I   1005.0);

// KZE14_V812103 SpI 029 Ventil
      CALL FC    14 (
           UnitNo                   := #UnitNo,
           SpIRec                   := DB2791.KZE14_V812103,
           SpIBit                   := I   1005.1);

NETWORK
TITLE =messages

      NOP   0;
// msg001 Msg 001 Message 01
      CALL FC    16 (
           UnitNo                   := #UnitNo,
           MsgRec                   := DB2797.msg001,
           MsgBit                   := DB2797.DBX   82.7);

// msg002 Msg 002 Message 02
      CALL FC    16 (
           UnitNo                   := #UnitNo,
           MsgRec                   := DB2797.msg002,
           MsgBit                   := DB2797.DBX  142.7);

// msg003 Msg 003 Message 03
      CALL FC    16 (
           UnitNo                   := #UnitNo,
           MsgRec                   := DB2797.msg003,
           MsgBit                   := DB2797.DBX  202.7);

NETWORK
TITLE =unit supply

      UC    FB [#UnitFB];
NETWORK
TITLE =KZE14_CIP_laeuft  A 1002.0 KZE14 CIP Läuft
// Act 002
// Box           : A14 KZE
// Output address: Q1002.0
      CALL FC    70 (
           UnitNo                   := #UnitNo,
           ActRec                   := DB2790.KZE14_CIP_laeuft,
           Typ                      := 0,
           FBa                      := #xTmp,
           FBa2                     := #xTmp,
           Out                      := Q   1002.0);

NETWORK
TITLE =KZE14_CIP_ENDE  A 1002.3 KZE14 CIP ENDE
// Act 003
// Box           : A14 KZE
// Output address: Q1002.3
      CALL FC    70 (
           UnitNo                   := #UnitNo,
           ActRec                   := DB2790.KZE14_CIP_ENDE,
           Typ                      := 0,
           FBa                      := #xTmp,
           FBa2                     := #xTmp,
           Out                      := Q   1002.3);

NETWORK
TITLE =KZE14_Abpumpen  A 1002.6 KZE14 Abpumpen
// Act 005
// Box           : A14 KZE
// Output address: Q1002.6
      CALL FC    70 (
           UnitNo                   := #UnitNo,
           ActRec                   := DB2790.KZE14_Abpumpen,
           Typ                      := 0,
           FBa                      := #xTmp,
           FBa2                     := #xTmp,
           Out                      := Q   1002.6);

NETWORK
TITLE =KZE14_KRSL_OA_PT  A 1002.4 KZE14 Kreislauf ohne Ablauf Puffertank
// Act 006
// Box           : A14 KZE
// Output address: Q1002.4
      CALL FC    70 (
           UnitNo                   := #UnitNo,
           ActRec                   := DB2790.KZE14_KRSL_OA_PT,
           Typ                      := 0,
           FBa                      := #xTmp,
           FBa2                     := #xTmp,
           Out                      := Q   1002.4);

NETWORK
TITLE =KZE14_KRSL_MA_PT  A 1002.5 KZE14 Kreislauf mit Ablauf Puffertank
// Act 007
// Box           : A14 KZE
// Output address: Q1002.5
      CALL FC    70 (
           UnitNo                   := #UnitNo,
           ActRec                   := DB2790.KZE14_KRSL_MA_PT,
           Typ                      := 0,
           FBa                      := #xTmp,
           FBa2                     := #xTmp,
           Out                      := Q   1002.5);

NETWORK
TITLE =KZE14_Grundstellung  A 1002.2 KZE14 Grundstellung
// Act 008
// Box           : A14 KZE
// Output address: Q1002.2
      CALL FC    70 (
           UnitNo                   := #UnitNo,
           ActRec                   := DB2790.KZE14_Grundstellung,
           Typ                      := 0,
           FBa                      := #xTmp,
           FBa2                     := #xTmp,
           Out                      := Q   1002.2);

NETWORK
TITLE =KZE14_Heizung_ein  A 1002.1 KZE14 Heizung ein
// Act 012
// Box           : A14 KZE
// Output address: Q1002.1
      CALL FC    70 (
           UnitNo                   := #UnitNo,
           ActRec                   := DB2790.KZE14_Heizung_ein,
           Typ                      := 0,
           FBa                      := #xTmp,
           FBa2                     := #xTmp,
           Out                      := Q   1002.1);

NETWORK
TITLE =KZE14_H2O  A 1003.1 KZE14 Hauptschritte Wasser
// Act 013
// Box           : A14 KZE
// Output address: Q1003.1
      CALL FC    70 (
           UnitNo                   := #UnitNo,
           ActRec                   := DB2790.KZE14_H2O,
           Typ                      := 0,
           FBa                      := #xTmp,
           FBa2                     := #xTmp,
           Out                      := Q   1003.1);

NETWORK
TITLE =KZE14_Lauge  A 1003.2 KZE14 Lauge Kreislauf
// Act 014
// Box           : A14 KZE
// Output address: Q1003.2
      CALL FC    70 (
           UnitNo                   := #UnitNo,
           ActRec                   := DB2790.KZE14_Lauge,
           Typ                      := 0,
           FBa                      := #xTmp,
           FBa2                     := #xTmp,
           Out                      := Q   1003.2);

NETWORK
TITLE =KZE14_Saeure  A 1003.3 KZE14 Säure Kreislauf
// Act 015
// Box           : A14 KZE
// Output address: Q1003.3
      CALL FC    70 (
           UnitNo                   := #UnitNo,
           ActRec                   := DB2790.KZE14_Saeure,
           Typ                      := 0,
           FBa                      := #xTmp,
           FBa2                     := #xTmp,
           Out                      := Q   1003.3);

NETWORK
TITLE =KZE14_Sterilisation  A 1003.4 KZE14 Sterilisation angewählt
// Act 016
// Box           : A14 KZE
// Output address: Q1003.4
      CALL FC    70 (
           UnitNo                   := #UnitNo,
           ActRec                   := DB2790.KZE14_Sterilisation,
           Typ                      := 0,
           FBa                      := #xTmp,
           FBa2                     := #xTmp,
           Out                      := Q   1003.4);

NETWORK
TITLE =KZE14_Abkuehlen  A 1003.5 KZE14 Abkühlen
// Act 017
// Box           : A14 KZE
// Output address: Q1003.5
      CALL FC    70 (
           UnitNo                   := #UnitNo,
           ActRec                   := DB2790.KZE14_Abkuehlen,
           Typ                      := 0,
           FBa                      := #xTmp,
           FBa2                     := #xTmp,
           Out                      := Q   1003.5);

END_FUNCTION_BLOCK

FUNCTION_BLOCK FB 1791
TITLE =U079: KZE Anlage 14
FAMILY : BOTEC_F1
NAME : U079E
VERSION : 1.2


VAR_TEMP
  CIP : BOOL ;	//CIP active
  UNIM : BOOL ;	//Unit Not In Maintenance
  GenRel : BOOL ;	//general OK (emergency and maintenance OK)
  EStopOK : BOOL ;	//emergency OK
  UnitNo : INT ;	//unit number
  xTmp : BOOL ;	//Temporary Bool
  iTmp : INT ;	//Temporary INT
  rTmp : REAL ;	//Temporary REAL
  dTmp : DINT ;	//Temporary DINT (free for general use)
  RetValInt : INT ;	//return value
END_VAR
BEGIN
NETWORK
TITLE =General

      SET   ;
// Simulation ---------------------------------------------------------------
      A     DB1791.DBX 1357.7;
      CC    FB  1799; // "U079Sim"
      A     DB1791.DBX   17.3;
      =     DB1791.DBX 1357.7; //Help bit for simulation

// get unit number ----------------------------------------------------------
      L     DB1790.DBW    0;
      T     #UnitNo;

// CIP ----------------------------------------------------------------------
      L     DB1791.DBD   54;
      L     0;
      <D    ;
      =     #CIP;

// emergency OK -------------------------------------------------------------
      A     DB1795.DBX   27.0; //Emergency Stop OK
      =     #EStopOK;

// Write Unit in Maintenance ------------------------------------------------

      AN    DB1791.DBX   69.7;
      =     #UNIM;

// emergency and maintenance OK ---------------------------------------------
      A     #EStopOK;
      A     #UNIM;
      =     #GenRel;

// communication ------------------------------------------------------------
      UC    FB  1795; // U079Com

NETWORK
TITLE =Analog Inputs

      NOP   0;

// ----------------------------------------------------------
// A14_KZE_FIC7101
// ----------------------------------------------------------

      L     ID  1006;
      T     DB2793.DBD  214;
      SET   ;
      =     DB2793.DBX  143.5;

      L     DB1791.DBD 1118; // !!! insert correct SFM !!!
      T     DB2793.DBD  238;

      SET   ;
      =     DB2793.DBX  141.5;

// ----------------------------------------------------------
// A14_KZE_TIR7101
// ----------------------------------------------------------

      L     ID  1010;
      T     DB2793.DBD  334;
      SET   ;
      =     DB2793.DBX  263.5;

      L     DB1791.DBD 1118; // !!! insert correct SFM !!!
      T     DB2793.DBD  358;

      SET   ;
      =     DB2793.DBX  261.5;

// ----------------------------------------------------------
// A14_KZE_TIC7102
// ----------------------------------------------------------

      L     ID  1014;
      T     DB2793.DBD  454;
      SET   ;
      =     DB2793.DBX  383.5;

      L     DB1791.DBD 1118; // !!! insert correct SFM !!!
      T     DB2793.DBD  478;

      SET   ;
      =     DB2793.DBX  381.5;

// ----------------------------------------------------------
// A14_KZE_CIS7102
// ----------------------------------------------------------

      L     ID  1018;
      T     DB2793.DBD  574;
      SET   ;
      =     DB2793.DBX  503.5;

      L     DB1791.DBD 1118; // !!! insert correct SFM !!!
      T     DB2793.DBD  598;

      SET   ;
      =     DB2793.DBX  501.5;

// ----------------------------------------------------------
// A14_KZE_TIS7111
// ----------------------------------------------------------

      L     ID  1022;
      T     DB2793.DBD  694;
      SET   ;
      =     DB2793.DBX  623.5;

      L     DB1791.DBD 1118; // !!! insert correct SFM !!!
      T     DB2793.DBD  718;

      SET   ;
      =     DB2793.DBX  621.5;


NETWORK
TITLE =Universal Value

      NOP   0;

// ----------------------------------------------------------
// unv001 Process Status
// ----------------------------------------------------------
// process value to UnV
//      L     0.000000e+000
//      T     "U079UnVD".unv001.ValExt

// ----------------------------------------------------------
// unv002 Universal Value 02
// ----------------------------------------------------------
// process value to UnV
//      L     0.000000e+000
//      T     "U079UnVD".unv002.ValExt

// ----------------------------------------------------------
// unv003 Universal Value 03
// ----------------------------------------------------------
// process value to UnV
//      L     0.000000e+000
//      T     "U079UnVD".unv003.ValExt

// ----------------------------------------------------------
// unv004 Universal Value 04
// ----------------------------------------------------------
// process value to UnV
//      L     0.000000e+000
//      T     "U079UnVD".unv004.ValExt

NETWORK
TITLE =Special Input

      NOP   0;

// ----------------------------------------------------------
// KZE14_CIP_BEREIT
// ----------------------------------------------------------
//      CLR
//      =     "U079SpID".KZE14_CIP_BEREIT.EAl
//      =     "U079SpID".KZE14_CIP_BEREIT.Pre

// ----------------------------------------------------------
// KZE14_PT_VOLL
// ----------------------------------------------------------
//      CLR
//      =     "U079SpID".KZE14_PT_VOLL.EAl
//      =     "U079SpID".KZE14_PT_VOLL.Pre

// ----------------------------------------------------------
// KZE14_PT_LEER
// ----------------------------------------------------------
//      CLR
//      =     "U079SpID".KZE14_PT_LEER.EAl
//      =     "U079SpID".KZE14_PT_LEER.Pre

// ----------------------------------------------------------
// KZE14_BEREIT_F_KREISL
// ----------------------------------------------------------
//      CLR
//      =     "U079SpID".KZE14_BEREIT_F_KREISL.EAl
//      =     "U079SpID".KZE14_BEREIT_F_KREISL.Pre

// ----------------------------------------------------------
// KZE14_STERI_BEREIT
// ----------------------------------------------------------
//      CLR
//      =     "U079SpID".KZE14_STERI_BEREIT.EAl
//      =     "U079SpID".KZE14_STERI_BEREIT.Pre

// ----------------------------------------------------------
// KZE14_AUSL_90GRAD
// ----------------------------------------------------------
//      CLR
//      =     "U079SpID".KZE14_AUSL_90GRAD.EAl
//      =     "U079SpID".KZE14_AUSL_90GRAD.Pre

// ----------------------------------------------------------
// KZE14_FRG_KZE Freigabe CIP nur KZE
// ----------------------------------------------------------
//      CLR
//      =     "U079SpID".KZE14_FRG_KZE.EAl
//      =     "U079SpID".KZE14_FRG_KZE.Pre

// ----------------------------------------------------------
// KZE14_FRG_MIX_KZE_FUEL Freigabe CIP Mixer KZE Füller
// ----------------------------------------------------------
//      CLR
//      =     "U079SpID".KZE14_FRG_MIX_KZE_FUEL.EAl
//      =     "U079SpID".KZE14_FRG_MIX_KZE_FUEL.Pre

// ----------------------------------------------------------
// KZE14_FRG_MIX_FUEL Freigabe CIP Mixer Füller
// ----------------------------------------------------------
//      CLR
//      =     "U079SpID".KZE14_FRG_MIX_FUEL.EAl
//      =     "U079SpID".KZE14_FRG_MIX_FUEL.Pre

// ----------------------------------------------------------
// KZE14_FRG_KZE_FUEL Freigabe CIP KZE Füller
// ----------------------------------------------------------
//      CLR
//      =     "U079SpID".KZE14_FRG_KZE_FUEL.EAl
//      =     "U079SpID".KZE14_FRG_KZE_FUEL.Pre

// ----------------------------------------------------------
// KZE14_V710021 Ventil
// ----------------------------------------------------------
//      CLR
//      =     "U079SpID".KZE14_V710021.EAl
//      =     "U079SpID".KZE14_V710021.Pre

// ----------------------------------------------------------
// KZE14_V710131 Ventil
// ----------------------------------------------------------
//      CLR
//      =     "U079SpID".KZE14_V710131.EAl
//      =     "U079SpID".KZE14_V710131.Pre

// ----------------------------------------------------------
// KZE14_V710005 Ventil
// ----------------------------------------------------------
//      CLR
//      =     "U079SpID".KZE14_V710005.EAl
//      =     "U079SpID".KZE14_V710005.Pre

// ----------------------------------------------------------
// KZE14_V710181 Ventil
// ----------------------------------------------------------
//      CLR
//      =     "U079SpID".KZE14_V710181.EAl
//      =     "U079SpID".KZE14_V710181.Pre

// ----------------------------------------------------------
// KZE14_V710182 Ventil
// ----------------------------------------------------------
//      CLR
//      =     "U079SpID".KZE14_V710182.EAl
//      =     "U079SpID".KZE14_V710182.Pre

// ----------------------------------------------------------
// KZE14_V813101 Ventil
// ----------------------------------------------------------
//      CLR
//      =     "U079SpID".KZE14_V813101.EAl
//      =     "U079SpID".KZE14_V813101.Pre

// ----------------------------------------------------------
// KZE14_V813102 Ventil
// ----------------------------------------------------------
//      CLR
//      =     "U079SpID".KZE14_V813102.EAl
//      =     "U079SpID".KZE14_V813102.Pre

// ----------------------------------------------------------
// KZE14_V812101 Ventil
// ----------------------------------------------------------
//      CLR
//      =     "U079SpID".KZE14_V812101.EAl
//      =     "U079SpID".KZE14_V812101.Pre

// ----------------------------------------------------------
// KZE14_V812102 Ventil
// ----------------------------------------------------------
//      CLR
//      =     "U079SpID".KZE14_V812102.EAl
//      =     "U079SpID".KZE14_V812102.Pre

// ----------------------------------------------------------
// KZE14_V812103 Ventil
// ----------------------------------------------------------
//      CLR
//      =     "U079SpID".KZE14_V812103.EAl
//      =     "U079SpID".KZE14_V812103.Pre

NETWORK
TITLE =Messages

      NOP   0;

// ----------------------------------------------------------
// msg001 Message 01
// ----------------------------------------------------------
      SET   ;
      R     DB2797.DBX   80.7;
      =     DB2797.DBX   81.4;

      CLR   ;
      =     DB2797.DBX   82.7;

// ----------------------------------------------------------
// msg002 Message 02
// ----------------------------------------------------------
      SET   ;
      R     DB2797.DBX  140.7;
      =     DB2797.DBX  141.4;

      CLR   ;
      =     DB2797.DBX  142.7;

// ----------------------------------------------------------
// msg003 Message 03
// ----------------------------------------------------------
      SET   ;
      R     DB2797.DBX  200.7;
      =     DB2797.DBX  201.4;

      CLR   ;
      =     DB2797.DBX  202.7;

NETWORK
TITLE =Sequence organisation

      CLR   ;
      =     M    122.2;

// SFM supply ----------------------------------------------------------------

// analog value to SFM  -----------------------
      L     DB2793.DBD  146;
      T     DB1791.DBD 1122; // !!! insert correct SFM !!!

// analog value to SFM  -----------------------
      L     DB2793.DBD  266;
      T     DB1791.DBD 1122; // !!! insert correct SFM !!!

// analog value to SFM  -----------------------
      L     DB2793.DBD  386;
      T     DB1791.DBD 1122; // !!! insert correct SFM !!!

// analog value to SFM  -----------------------
      L     DB2793.DBD  506;
      T     DB1791.DBD 1122; // !!! insert correct SFM !!!

// analog value to SFM  -----------------------
      L     DB2793.DBD  626;
      T     DB1791.DBD 1122; // !!! insert correct SFM !!!

// sequencer ----------------------------------------------------------------
      A     DB1793.DBX   43.1;
      S     DB1793.DBX   97.3;

      CALL FC    40 (
           UnitNo                   := #UnitNo);

NETWORK
TITLE =Auto / Manual

      SET   ;
      AN    M    122.2;
      JC    MODE;
      AN    M    120.1;

// assign actuator mode
      AN    M    120.1;
      =     DB2790.DBX  185.4;
      =     DB2790.DBX  265.4;
      =     DB2790.DBX  425.4;
      =     DB2790.DBX  505.4;
      =     DB2790.DBX  585.4;
      =     DB2790.DBX  665.4;
      =     DB2790.DBX  985.4;
      =     DB2790.DBX 1065.4;
      =     DB2790.DBX 1145.4;
      =     DB2790.DBX 1225.4;
      =     DB2790.DBX 1305.4;
      =     DB2790.DBX 1385.4;



MODE: SET   ;

NETWORK
TITLE =KZE14_CIP_laeuft A 1002.0 KZE14 CIP Läuft
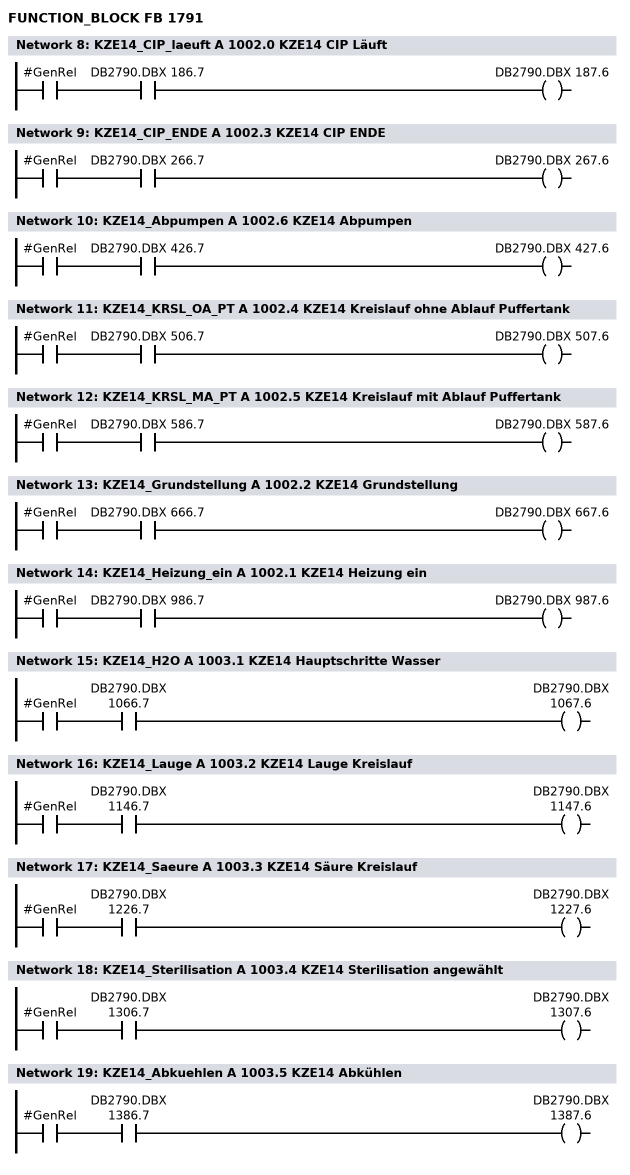

      A     #GenRel;
      A     DB2790.DBX  186.7;
      =     DB2790.DBX  187.6;
NETWORK
TITLE =KZE14_CIP_ENDE A 1002.3 KZE14 CIP ENDE

      A     #GenRel;
      A     DB2790.DBX  266.7;
      =     DB2790.DBX  267.6;
NETWORK
TITLE =KZE14_Abpumpen A 1002.6 KZE14 Abpumpen

      A     #GenRel;
      A     DB2790.DBX  426.7;
      =     DB2790.DBX  427.6;
NETWORK
TITLE =KZE14_KRSL_OA_PT A 1002.4 KZE14 Kreislauf ohne Ablauf Puffertank

      A     #GenRel;
      A     DB2790.DBX  506.7;
      =     DB2790.DBX  507.6;
NETWORK
TITLE =KZE14_KRSL_MA_PT A 1002.5 KZE14 Kreislauf mit Ablauf Puffertank

      A     #GenRel;
      A     DB2790.DBX  586.7;
      =     DB2790.DBX  587.6;
NETWORK
TITLE =KZE14_Grundstellung A 1002.2 KZE14 Grundstellung

      A     #GenRel;
      A     DB2790.DBX  666.7;
      =     DB2790.DBX  667.6;
NETWORK
TITLE =KZE14_Heizung_ein A 1002.1 KZE14 Heizung ein

      A     #GenRel;
      A     DB2790.DBX  986.7;
      =     DB2790.DBX  987.6;
NETWORK
TITLE =KZE14_H2O A 1003.1 KZE14 Hauptschritte Wasser

      A     #GenRel;
      A     DB2790.DBX 1066.7;
      =     DB2790.DBX 1067.6;
NETWORK
TITLE =KZE14_Lauge A 1003.2 KZE14 Lauge Kreislauf

      A     #GenRel;
      A     DB2790.DBX 1146.7;
      =     DB2790.DBX 1147.6;
NETWORK
TITLE =KZE14_Saeure A 1003.3 KZE14 Säure Kreislauf

      A     #GenRel;
      A     DB2790.DBX 1226.7;
      =     DB2790.DBX 1227.6;
NETWORK
TITLE =KZE14_Sterilisation A 1003.4 KZE14 Sterilisation angewählt

      A     #GenRel;
      A     DB2790.DBX 1306.7;
      =     DB2790.DBX 1307.6;
NETWORK
TITLE =KZE14_Abkuehlen A 1003.5 KZE14 Abkühlen

      A     #GenRel;
      A     DB2790.DBX 1386.7;
      =     DB2790.DBX 1387.6;
END_FUNCTION_BLOCK

FUNCTION_BLOCK FB 1810
TITLE =U081: Caustic Tank
FAMILY : BOTEC_F1
NAME : UniA
VERSION : 2.1


VAR_TEMP
  EStopOK : BOOL ;	//auxiliary flag
  CIP : BOOL ;	//CIP Program Selected
  xTmp : BOOL ;	//Temporary Bool(free for general use)
  UnitNo : INT ;	//unit number
  UnitFB : INT ;	//unit expansion FB number
  rTmp : REAL ;	//Temporary REAL (free for general use)
  iTmp : INT ;	//Temporary INT (free for general use)
  dTmp : DINT ;	//Temporary DINT (free for general use)
END_VAR
BEGIN
NETWORK
TITLE =general

      CLR   ;
      =     #xTmp;
      =     #EStopOK;

      L     DB1810.DBW    0;
      T     #UnitNo;
      L     DB1810.DBW    2;
      T     #UnitFB;

NETWORK
TITLE =analog inputs

      NOP   0;
// LI_L AnI 001 Laugetank
      CALL FC    24 (
           UnitNo                   := #UnitNo,
           AnIRec                   := DB2813.LI_L,
           ValPer                   := IW   566);

// CS_L AnI 002 Laugetank
      CALL FC    24 (
           UnitNo                   := #UnitNo,
           AnIRec                   := DB2813.CS_L,
           ValPer                   := IW   154);

NETWORK
TITLE =Universal value

      NOP   0;
// unv001 UnV 001 Process Status
      CALL FC    27 (
           UnitNo                   := #UnitNo,
           UnVRec                   := DB2815.unv001,
           ValExt                   := DB2815.DBD  234);

// unv002 UnV 002 Universal Value 02
      CALL FC    27 (
           UnitNo                   := #UnitNo,
           UnVRec                   := DB2815.unv002,
           ValExt                   := DB2815.DBD  362);

NETWORK
TITLE =special inputs

      NOP   0;
// LS_LLL_LAUGE SpI 001 Laugetank LS-
      CALL FC    14 (
           UnitNo                   := #UnitNo,
           SpIRec                   := DB2811.LS_LLL_LAUGE,
           SpIBit                   := I     92.2);

// LS_HL_LAUGE SpI 002 Laugetank LS+
      CALL FC    14 (
           UnitNo                   := #UnitNo,
           SpIRec                   := DB2811.LS_HL_LAUGE,
           SpIBit                   := I     92.0);

// LS_LL_LAUGE SpI 003 Laugetank LS/
      CALL FC    14 (
           UnitNo                   := #UnitNo,
           SpIRec                   := DB2811.LS_LL_LAUGE,
           SpIBit                   := I      7.3);

// LS_LL_LAUGE_ALT SpI 004 Spare
//      CALL  "SI1"
//       UnitNo:=#UnitNo
//       SpIRec:="U081SpID".LS_LL_LAUGE_ALT
//       SpIBit:="LS_LL_LAUGE_ALT"

// U81_SpI005 SpI 005 spare
//      CALL  "SI1"
//       UnitNo:=#UnitNo
//       SpIRec:="U081SpID".U81_SpI005
//       SpIBit:=#xTmp

// LANG_NEUANSATZ_LAUGE SpI 007 RUECKMELDUNG VON LANG AN TU
      CALL FC    14 (
           UnitNo                   := #UnitNo,
           SpIRec                   := DB2811.LANG_NEUANSATZ_LAUGE,
           SpIBit                   := I     40.0);

// LANG_NACHSCH_LAUGE SpI 008 RUECKMELDUNG VON LANG AN TU
      CALL FC    14 (
           UnitNo                   := #UnitNo,
           SpIRec                   := DB2811.LANG_NACHSCH_LAUGE,
           SpIBit                   := I     40.4);

NETWORK
TITLE =messages

      NOP   0;
// msg001 Msg 001 Message 01
      CALL FC    16 (
           UnitNo                   := #UnitNo,
           MsgRec                   := DB2817.msg001,
           MsgBit                   := DB2817.DBX   82.7);

// msg002 Msg 002 Message 02
      CALL FC    16 (
           UnitNo                   := #UnitNo,
           MsgRec                   := DB2817.msg002,
           MsgBit                   := DB2817.DBX  142.7);

NETWORK
TITLE =unit supply

      UC    FB [#UnitFB];

NETWORK
TITLE =RW_LAUGE  Rührwerk HLT
// Act 001
// Box           : LT-CIP
// Input address : I256.2
// Output address: Q256.2
      CALL FC    70 (
           UnitNo                   := #UnitNo,
           ActRec                   := DB2810.RW_LAUGE,
           Typ                      := 1,
           FBa                      := #xTmp,
           FBa2                     := I    256.2,
           Out                      := Q    256.2);

NETWORK
TITLE =LU_P1  LUP1
// Act 002
// Box           : S6 U6.3
// Input address : I5.5
// Output address: Q5.5
//      CALL  "Act"
//       UnitNo:=#UnitNo
//       ActRec:="U081ActD".LU_P1
//       Typ   :=0
//       FBa   :="LU_P1GSK"
//       FBa2  :=#xTmp
//       Out   :="LU_P1O"

NETWORK
TITLE =U81_Act003  spare
// Act 003
// Box           :
// Input address : #xTmp
// Output address: #xTmp
//      CALL  "Act"
//       UnitNo:=#UnitNo
//       ActRec:="U081ActD".U81_Act003
//       Typ   :=3
//       FBa   :=#xTmp
//       FBa2  :=#xTmp
//       Out   :=#xTmp

NETWORK
TITLE =U81_Act004  Säure Umpumpvetil
// Act 004
// Box           :
// Input address : #xTmp
// Output address: #xTmp
//      CALL  "Act"
//       UnitNo:=#UnitNo
//       ActRec:="U081ActD".U81_Act004
//       Typ   :=0
//       FBa   :=#xTmp
//       FBa2  :="SU_K1GSC"
//       Out   :="SU_K1O"

NETWORK
TITLE =U81_Act005  spare
// Act 005
// Box           :
// Input address : #xTmp
// Output address: #xTmp
//      CALL  "Act"
//       UnitNo:=#UnitNo
//       ActRec:="U081ActD".U81_Act005
//       Typ   :=3
//       FBa   :=#xTmp
//       FBa2  :=#xTmp
//       Out   :=#xTmp

NETWORK
TITLE =U81_Act006  spare
// Act 006
// Box           :
// Input address : #xTmp
// Output address: #xTmp
//      CALL  "Act"
//       UnitNo:=#UnitNo
//       ActRec:="U081ActD".U81_Act006
//       Typ   :=3
//       FBa   :=#xTmp
//       FBa2  :=#xTmp
//       Out   :=#xTmp

NETWORK
TITLE =LU_K1  Lauge Umpumpventil
// Act 007
// Box           : VSRVK1..3
// Input address : I275.4
// Output address: Q275.4
      CALL FC    70 (
           UnitNo                   := #UnitNo,
           ActRec                   := DB2810.LU_K1,
           Typ                      := 1,
           FBa                      := #xTmp,
           FBa2                     := I    275.4,
           Out                      := Q    275.4);

NETWORK
TITLE =LANGF_NACHSCHLAUGE  SIGNAL VON TU AN FA.LANG
// Act 008
// Box           : S8 U8.2
// Output address: Q43.0
      CALL FC    70 (
           UnitNo                   := #UnitNo,
           ActRec                   := DB2810.LANGF_NACHSCHLAUGE,
           Typ                      := 0,
           FBa                      := #xTmp,
           FBa2                     := #xTmp,
           Out                      := Q     43.0);

NETWORK
TITLE =LANGF_NEUANSLAUGE  SIGNAL VON TU AN FA.LANG
// Act 009
// Box           : S8 U8.2
// Output address: Q43.3
      CALL FC    70 (
           UnitNo                   := #UnitNo,
           ActRec                   := DB2810.LANGF_NEUANSLAUGE,
           Typ                      := 0,
           FBa                      := #xTmp,
           FBa2                     := #xTmp,
           Out                      := Q     43.3);

END_FUNCTION_BLOCK

FUNCTION_BLOCK FB 1811
TITLE =U081: Caustic Tank
FAMILY : BOTEC_F1
NAME : UniE
VERSION : 1.2


VAR_TEMP
  CIP : BOOL ;	//CIP active
  UNIM : BOOL ;	//Unit Not In Maintenance
  GenRel : BOOL ;	//general OK (emergency and maintenance OK)
  EStopOK : BOOL ;	//emergency OK
  UnitNo : INT ;	//unit number
  xTmp : BOOL ;	//Temporary Bool
  iTmp : INT ;	//Temporary INT
  rTmp : REAL ;	//Temporary REAL
  dTmp : DINT ;	//Temporary DINT (free for general use)
  RetValInt : INT ;	//return value
END_VAR
BEGIN
NETWORK
TITLE =General

      SET   ;
// Simulation ---------------------------------------------------------------
      A     DB1811.DBX 1357.7;
      CC    FB  1819; // "U081Sim"
      A     DB1811.DBX   17.3;
      =     DB1811.DBX 1357.7; //Help bit for simulation

// get unit number ----------------------------------------------------------
      L     DB1810.DBW    0;
      T     #UnitNo;

// CIP ----------------------------------------------------------------------
      L     DB1811.DBD   54;
      L     0;
      <D    ;
      =     #CIP;

// emergency OK -------------------------------------------------------------
      A     DB1815.DBX   27.0; //Emergency Stop OK
      =     #EStopOK;

// Write Unit in Maintenance ------------------------------------------------

      AN    DB1811.DBX   69.7;
      =     #UNIM;

// emergency and maintenance OK ---------------------------------------------
      A     #EStopOK;
      A     #UNIM;
      =     #GenRel;

// communication ------------------------------------------------------------
      UC    FB  1815; // U081Com

NETWORK
TITLE =Analog Inputs

      NOP   0;

// ----------------------------------------------------------
// LI_L Laugetank
// ----------------------------------------------------------
      L     DB1811.DBD 1118; // !!! insert correct SFM !!!
      T     DB2813.DBD  238;

//      SET
//      =     "U081AnID".LI_L.EAlHH

// ----------------------------------------------------------
// CS_L Laugetank
// ----------------------------------------------------------
      L     DB1811.DBD 1118; // !!! insert correct SFM !!!
      T     DB2813.DBD  358;

      SET   ;
      =     DB2813.DBX  261.5;

NETWORK
TITLE =Universal Value

      NOP   0;

// ----------------------------------------------------------
// unv001 Process Status
// ----------------------------------------------------------
// process value to UnV
//      L     0.000000e+000
//      T     "U081UnVD".unv001.ValExt

// ----------------------------------------------------------
// unv002 Universal Value 02
// ----------------------------------------------------------
// process value to UnV
//      L     0.000000e+000
//      T     "U081UnVD".unv002.ValExt

NETWORK
TITLE =Special Input

      NOP   0;

// ----------------------------------------------------------
// LS_LLL_LAUGE Laugetank LS-
// ----------------------------------------------------------
      ON    DB2910.DBX  662.5;
      ON    DB2920.DBX  662.5;
      ON    DB2930.DBX  662.5;
      =     DB2811.DBX   81.4;

      CLR   ;
      =     DB2811.DBX   81.5;

// ----------------------------------------------------------
// LS_HL_LAUGE Laugetank LS+
// ----------------------------------------------------------
      ON    DB2910.DBX  742.5;
      ON    DB2920.DBX  742.5;
      ON    DB2930.DBX  742.5;
      =     DB2811.DBX  141.4;
      SET   ;
      =     DB2811.DBX  141.5;

      SET   ;
      =     DB2811.DBX  140.6;

// ----------------------------------------------------------
// LS_LL_LAUGE Laugetank LS/
// ----------------------------------------------------------
      CLR   ;
//      =     "U081SpID".LS_LL_LAUGE.EAl
      =     DB2811.DBX  201.5;

// ----------------------------------------------------------
// LS_LL_LAUGE_ALT
// ----------------------------------------------------------
      CLR   ;
      =     DB2811.DBX  261.4;
      =     DB2811.DBX  261.5;

// ----------------------------------------------------------
// U81_SpI005 spare
// ----------------------------------------------------------
      CLR   ;
      =     DB2811.DBX  321.4;
      =     DB2811.DBX  321.5;

// ----------------------------------------------------------
// LANG_NEUANSATZ_LAUGE RUECKMELDUNG VON LANG AN TU
// ----------------------------------------------------------
      CLR   ;
//      =     "U081SpID".LANG_NEUANSATZ_LAUGE.EAl
//      =     "U081SpID".LANG_NEUANSATZ_LAUGE.Pre

// ----------------------------------------------------------
// LANG_NACHSCH_LAUGE RUECKMELDUNG VON LANG AN TU
// ----------------------------------------------------------
      CLR   ;
//      =     "U081SpID".LANG_NACHSCH_LAUGE.EAl
//      =     "U081SpID".LANG_NACHSCH_LAUGE.Pre

NETWORK
TITLE =Messages

      NOP   0;

// ----------------------------------------------------------
// msg001 Message 01
// ----------------------------------------------------------
      SET   ;
      R     DB2817.DBX   80.7;
      =     DB2817.DBX   81.4;

      CLR   ;
      =     DB2817.DBX   82.7;

// ----------------------------------------------------------
// msg002 Message 02
// ----------------------------------------------------------
      SET   ;
      R     DB2817.DBX  140.7;
      =     DB2817.DBX  141.4;

      CLR   ;
      =     DB2817.DBX  142.7;

NETWORK
TITLE =Sequence organisation

      CLR   ;
      =     M    122.2;

// SFM supply ----------------------------------------------------------------

// analog value to SFM Laugetank -----------------------
      L     DB2813.DBD  146;
      T     DB1811.DBD  386; // Level

// analog value to SFM Laugetank -----------------------
      L     DB2813.DBD  266;
      T     DB1811.DBD  642; // Conductivity
      T     DB1811.DBD  658; // Conductivity Start Pulse/Pause

// sequencer ----------------------------------------------------------------
      A     DB1813.DBX   43.1;
      S     DB1813.DBX   97.3;

      CALL FC    40 (
           UnitNo                   := #UnitNo);

NETWORK
TITLE =Auto / Manual

      SET   ;
      AN    M    122.2;
      JC    MODE;
      AN    M    120.1;

// assign actuator mode
      AN    M    120.1;
      =     DB2810.DBX  105.4;
      =     DB2810.DBX  185.4;
      =     DB2810.DBX  265.4;
      =     DB2810.DBX  345.4;
      =     DB2810.DBX  425.4;
      =     DB2810.DBX  505.4;
      =     DB2810.DBX  585.4;
      =     DB2810.DBX  665.4;
      =     DB2810.DBX  745.4;



MODE: SET   ;

NETWORK
TITLE =RW_LAUGE Rührwerk HLT
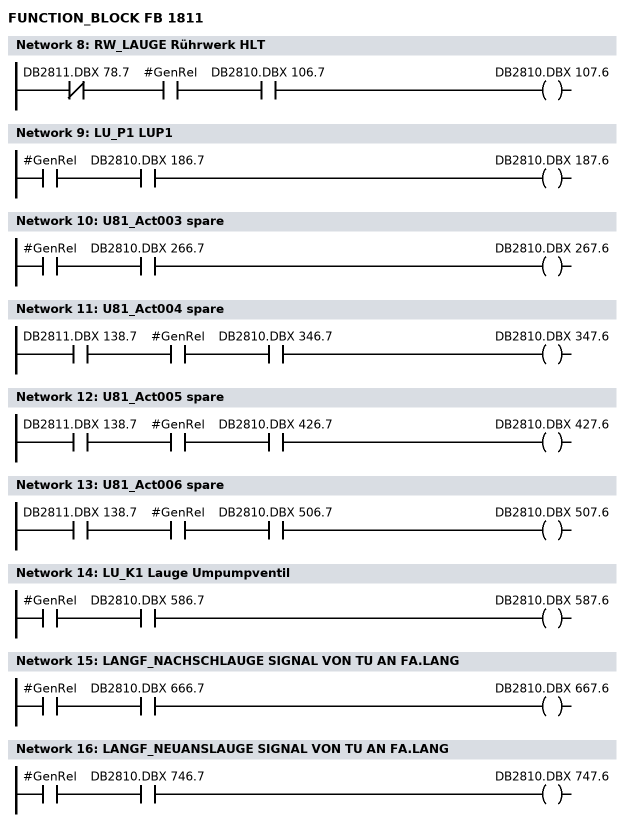

      AN    DB2811.DBX   78.7;
      A     #GenRel;
      A     DB2810.DBX  106.7;
      =     DB2810.DBX  107.6;
NETWORK
TITLE =LU_P1 LUP1

      A     #GenRel;
      A     DB2810.DBX  186.7;
      =     DB2810.DBX  187.6;
NETWORK
TITLE =U81_Act003 spare

      A     #GenRel;
      A     DB2810.DBX  266.7;
      =     DB2810.DBX  267.6;
NETWORK
TITLE =U81_Act004 spare

      A     DB2811.DBX  138.7;

      A     #GenRel;
      A     DB2810.DBX  346.7;
      =     DB2810.DBX  347.6;
NETWORK
TITLE =U81_Act005 spare

      A     DB2811.DBX  138.7;

      A     #GenRel;
      A     DB2810.DBX  426.7;
      =     DB2810.DBX  427.6;
NETWORK
TITLE =U81_Act006 spare

      A     DB2811.DBX  138.7;

      A     #GenRel;
      A     DB2810.DBX  506.7;
      =     DB2810.DBX  507.6;
NETWORK
TITLE =LU_K1 Lauge Umpumpventil

      A     #GenRel;
      A     DB2810.DBX  586.7;
      =     DB2810.DBX  587.6;
NETWORK
TITLE =LANGF_NACHSCHLAUGE SIGNAL VON TU AN FA.LANG

      A     #GenRel;
      A     DB2810.DBX  666.7;
      =     DB2810.DBX  667.6;
NETWORK
TITLE =LANGF_NEUANSLAUGE SIGNAL VON TU AN FA.LANG

      A     #GenRel;
      A     DB2810.DBX  746.7;
      =     DB2810.DBX  747.6;
END_FUNCTION_BLOCK

FUNCTION_BLOCK FB 1820
TITLE =U082: Acid Tank
FAMILY : BOTEC_F1
NAME : UniA
VERSION : 2.1


VAR_TEMP
  EStopOK : BOOL ;	//auxiliary flag
  CIP : BOOL ;	//CIP Program Selected
  xTmp : BOOL ;	//Temporary Bool(free for general use)
  UnitNo : INT ;	//unit number
  UnitFB : INT ;	//unit expansion FB number
  rTmp : REAL ;	//Temporary REAL (free for general use)
  iTmp : INT ;	//Temporary INT (free for general use)
  dTmp : DINT ;	//Temporary DINT (free for general use)
END_VAR
BEGIN
NETWORK
TITLE =general

      CLR   ;
      =     #xTmp;
      =     #EStopOK;

      L     DB1820.DBW    0;
      T     #UnitNo;
      L     DB1820.DBW    2;
      T     #UnitFB;

NETWORK
TITLE =analog inputs

      NOP   0;
// LI_S AnI 001 Säuretank
      CALL FC    24 (
           UnitNo                   := #UnitNo,
           AnIRec                   := DB2823.LI_S,
           ValPer                   := IW   564);

// CS_S AnI 002 Säuretank
      CALL FC    24 (
           UnitNo                   := #UnitNo,
           AnIRec                   := DB2823.CS_S,
           ValPer                   := IW   156);

NETWORK
TITLE =Universal value

      NOP   0;
// unv001 UnV 001 Process Status
      CALL FC    27 (
           UnitNo                   := #UnitNo,
           UnVRec                   := DB2825.unv001,
           ValExt                   := DB2825.DBD  234);

// unv002 UnV 002 Universal Value 02
      CALL FC    27 (
           UnitNo                   := #UnitNo,
           UnVRec                   := DB2825.unv002,
           ValExt                   := DB2825.DBD  362);

NETWORK
TITLE =special inputs

      NOP   0;
// LS_LLL_SAEURE SpI 001 Säuretank LS-
      CALL FC    14 (
           UnitNo                   := #UnitNo,
           SpIRec                   := DB2821.LS_LLL_SAEURE,
           SpIBit                   := I     92.7);

// LS_HL_SAEURE SpI 002 Säuretank LS+
      CALL FC    14 (
           UnitNo                   := #UnitNo,
           SpIRec                   := DB2821.LS_HL_SAEURE,
           SpIBit                   := I     92.5);

// LS_LL_SAEURE SpI 003 Säuretank LS/
      CALL FC    14 (
           UnitNo                   := #UnitNo,
           SpIRec                   := DB2821.LS_LL_SAEURE,
           SpIBit                   := I      7.4);

// LS_LL_SAEURE_ALT SpI 004 Spare
//      CALL  "SI1"
//       UnitNo:=#UnitNo
//       SpIRec:="U082SpID".LS_LL_SAEURE_ALT
//       SpIBit:="LS_LL_SAEURE_ALT"

// LANG_NEUANSATZ_SAEURE SpI 007 RUECKMELDUNG VON LANG AN TU
      CALL FC    14 (
           UnitNo                   := #UnitNo,
           SpIRec                   := DB2821.LANG_NEUANSATZ_SAEURE,
           SpIBit                   := I     40.1);

// LANG_NACHSCH_SAEURE SpI 008 RUECKMELDUNG VON LANG AN TU
      CALL FC    14 (
           UnitNo                   := #UnitNo,
           SpIRec                   := DB2821.LANG_NACHSCH_SAEURE,
           SpIBit                   := I     40.5);

NETWORK
TITLE =messages

      NOP   0;
// msg001 Msg 001 Message 01
      CALL FC    16 (
           UnitNo                   := #UnitNo,
           MsgRec                   := DB2827.msg001,
           MsgBit                   := DB2827.DBX   82.7);

// msg002 Msg 002 Message 02
      CALL FC    16 (
           UnitNo                   := #UnitNo,
           MsgRec                   := DB2827.msg002,
           MsgBit                   := DB2827.DBX  142.7);

NETWORK
TITLE =unit supply

      UC    FB [#UnitFB];

NETWORK
TITLE =RW_SAEURE  Rührwerk S1T
// Act 001
// Box           : LT-CIP
// Input address : I256.3
// Output address: Q256.3
      CALL FC    70 (
           UnitNo                   := #UnitNo,
           ActRec                   := DB2820.RW_SAEURE,
           Typ                      := 1,
           FBa                      := #xTmp,
           FBa2                     := I    256.3,
           Out                      := Q    256.3);

NETWORK
TITLE =SU_P1  SUP1
// Act 002
// Box           : S6 U6.3
// Input address : I5.6
// Output address: Q5.6
//      CALL  "Act"
//       UnitNo:=#UnitNo
//       ActRec:="U082ActD".SU_P1
//       Typ   :=0
//       FBa   :="SU_P1GSK"
//       FBa2  :=#xTmp
//       Out   :="SU_P1O"

NETWORK
TITLE =U82_Act004  spare
// Act 004
// Box           :
// Input address : #xTmp
// Output address: #xTmp
//      CALL  "Act"
//       UnitNo:=#UnitNo
//       ActRec:="U082ActD".U82_Act004
//       Typ   :=3
//       FBa   :=#xTmp
//       FBa2  :=#xTmp
//       Out   :=#xTmp

NETWORK
TITLE =U82_Act005  spare
// Act 005
// Box           :
// Input address : #xTmp
// Output address: #xTmp
//      CALL  "Act"
//       UnitNo:=#UnitNo
//       ActRec:="U082ActD".U82_Act005
//       Typ   :=3
//       FBa   :=#xTmp
//       FBa2  :=#xTmp
//       Out   :=#xTmp

NETWORK
TITLE =SU_K1  Säure Umpumpventil
// Act 007
// Box           : VSRVK1..3
// Input address : I275.5
// Output address: Q275.5
      CALL FC    70 (
           UnitNo                   := #UnitNo,
           ActRec                   := DB2820.SU_K1,
           Typ                      := 1,
           FBa                      := #xTmp,
           FBa2                     := I    275.5,
           Out                      := Q    275.5);

NETWORK
TITLE =LANGF_NACHSCHSAEURE  SIGNAL VON TU AN FA.LANG
// Act 008
// Box           : S8 U8.2
// Output address: Q43.1
      CALL FC    70 (
           UnitNo                   := #UnitNo,
           ActRec                   := DB2820.LANGF_NACHSCHSAEURE,
           Typ                      := 0,
           FBa                      := #xTmp,
           FBa2                     := #xTmp,
           Out                      := Q     43.1);

NETWORK
TITLE =LANGF_NEUANSSAEURE  SIGNAL VON TU AN FA.LANG
// Act 009
// Box           : S8 U8.2
// Output address: Q43.4
      CALL FC    70 (
           UnitNo                   := #UnitNo,
           ActRec                   := DB2820.LANGF_NEUANSSAEURE,
           Typ                      := 0,
           FBa                      := #xTmp,
           FBa2                     := #xTmp,
           Out                      := Q     43.4);

END_FUNCTION_BLOCK

FUNCTION_BLOCK FB 1821
TITLE =U082: Acid Tank
FAMILY : BOTEC_F1
NAME : UniE
VERSION : 1.2


VAR_TEMP
  CIP : BOOL ;	//CIP active
  UNIM : BOOL ;	//Unit Not In Maintenance
  GenRel : BOOL ;	//general OK (emergency and maintenance OK)
  EStopOK : BOOL ;	//emergency OK
  UnitNo : INT ;	//unit number
  xTmp : BOOL ;	//Temporary Bool
  iTmp : INT ;	//Temporary INT
  rTmp : REAL ;	//Temporary REAL
  dTmp : DINT ;	//Temporary DINT (free for general use)
  RetValInt : INT ;	//return value
END_VAR
BEGIN
NETWORK
TITLE =General

      SET   ;
// Simulation ---------------------------------------------------------------
      A     DB1821.DBX 1357.7;
      CC    FB  1829; // "U082Sim"
      A     DB1821.DBX   17.3;
      =     DB1821.DBX 1357.7; //Help bit for simulation

// get unit number ----------------------------------------------------------
      L     DB1820.DBW    0;
      T     #UnitNo;

// CIP ----------------------------------------------------------------------
      L     DB1821.DBD   54;
      L     0;
      <D    ;
      =     #CIP;

// emergency OK -------------------------------------------------------------
      A     DB1825.DBX   27.0; //Emergency Stop OK
      =     #EStopOK;

// Write Unit in Maintenance ------------------------------------------------

      AN    DB1821.DBX   69.7;
      =     #UNIM;

// emergency and maintenance OK ---------------------------------------------
      A     #EStopOK;
      A     #UNIM;
      =     #GenRel;

// communication ------------------------------------------------------------
      UC    FB  1825; // U082Com

NETWORK
TITLE =Analog Inputs

      NOP   0;

